(* PLC project LMM.project, Inovance company InoProShop(V1.9.1.6) InoProShop(V1.9.1.6) *)
(* stored: creationDateTime 2026-09-12T22:49:48.5577606, modificationDateTime 2026-09-12T22:49:26.9924488 *)

VAR_GLOBAL  (* GVL *)
  StartBtn AT %IX1.6 : BOOL;  (* 【面板启动】→ HMI_xStart *)
  StopBtn AT %IX1.4 : BOOL;  (* 【面板停止】→ HMI_xStop *)
  ResetBtn : BOOL;  (* 【面板复位】→ HMI_xStopHold3s；地址现场另绑 *)
  EStop AT %IX0.4 : BOOL;  (* 【面板急停】正常=TRUE 按下=FALSE *)
  StopLamp AT %QX0.6 : BOOL;  (* 【停止指示灯】← Dev_xStop *)
  StartLamp AT %QX0.7 : BOOL;  (* 【运行指示灯】← Dev_xRun *)
  JogFwd : BOOL;  (* 【面板前进】手动 X+ *)
  JogBwd : BOOL;  (* 【面板后退】手动 X- *)
  JogRight : BOOL;  (* 【面板右】手动 Y+ *)
  JogLeft : BOOL;  (* 【面板左】手动 Y- *)
  JogUp : BOOL;  (* 【面板上】手动 Z+ *)
  JogDown : BOOL;  (* 【面板下】手动 Z- *)
  JogClockAdd : BOOL;  (* 【面板顺时针】手动 R+ *)
  JogClockMis : BOOL;  (* 【面板逆时针】手动 R- *)
  HMI_xEStop : BOOL;  (* 【急停】TRUE正常 FALSE按下 = 物理 AND 触摸屏Req AND Web *)
  HMI_xStop : BOOL;  (* 【停止】任一源为真即停；长按3s=复位 *)
  HMI_xStopHold3s : BOOL;  (* 【复位】清急停锁存 + 轴故障复位 *)
  HMI_xStart : BOOL;  (* 【启动】上升沿 *)
  HMI_xEnable : BOOL;  (* 【启动别名】与 HMI_xStart 等效 *)
  xEStopLatched : BOOL;  (* 【急停锁存】仅复位可清 *)
  xFaultAggregate : BOOL;  (* 【故障汇总】任轴 ErrorStop *)
  eCtrlSrc : INT;  (* 【控制源】0=面板/触摸屏 1=远程Web；仅 PRG_TcpHmi 写 *)
  eOpMode : INT;  (* 【运行方式】0手动 1自动 *)
  iAlarmID : INT;  (* 【内部报警号】 *)
  HMI_eDevState : INT;  (* 【只读·状态码】0停 1运行 2错误 *)
  HMI_eOpMode : INT;  (* 【只读·方式显示】0手动 1自动 *)
  HMI_iAlarmShow : INT;  (* 【只读·报警号】1001急停 1002轴故障 1005力超时 1006从站失败 1007未就绪；1008已废 *)
  Dev_xStop : BOOL;  (* 【内部·停止派生】 *)
  Dev_xRun : BOOL;  (* 【内部·运行派生】 *)
  Dev_xError : BOOL;  (* 【内部·故障派生】 *)
  HMI_xDevStop : BOOL;  (* 【只读·停止灯】 *)
  HMI_xDevRun : BOOL;  (* 【只读·运行灯】 *)
  HMI_xDevError : BOOL;  (* 【只读·故障灯】 *)
  HMI_xLampEStop : BOOL;  (* 【只读·急停指示】 *)
  HMI_xLampEnableOk : BOOL;  (* 【只读·就绪灯】 *)
  HMI_xLampFault : BOOL;  (* 【只读·故障指示】 *)
  HMI_xAutoMode : BOOL;  (* 【模式】FALSE手动 TRUE自动 *)
  HMI_xJogXPos : BOOL;  (* 【X+】M1=M2 同速同向；与旋转互斥 *)
  HMI_xJogXNeg : BOOL;  (* 【X-】 *)
  HMI_xSpinLeft : BOOL;  (* 【左旋转】差速原地转；与 X± 互斥 *)
  HMI_xSpinRight : BOOL;  (* 【右旋转】 *)
  HMI_xJogYPos : BOOL;  (* 【Y+】受限位 *)
  HMI_xJogYNeg : BOOL;  (* 【Y-】 *)
  HMI_xJogZPos : BOOL;  (* 【Z+】回零后软限位 [-0.7,0] *)
  HMI_xJogZNeg : BOOL;  (* 【Z-】 *)
  HMI_xJogRPos : BOOL;  (* 【R+】需 xM5Ready *)
  HMI_xJogRNeg : BOOL;  (* 【R-】 *)
  HMI_xHomeY : BOOL;  (* 【Y回零】 *)
  HMI_xHomeZ : BOOL;  (* 【Z回零】完成后软限位生效 *)
  HMI_xHomeR : BOOL;  (* 【R回零】编码器回零 *)
  HMI_iHomeAxis : INT := 0;  (* 【回零轴选择】0无 1Y 2Z 3R *)
  HMI_xHomeExec : BOOL;  (* 【回零执行】对选定轴 *)
  HMI_xHomedY : BOOL;  (* 【只读·Y已回零】 *)
  HMI_xHomedZ : BOOL;  (* 【只读·Z已回零】 *)
  HMI_xHomedR : BOOL;  (* 【只读·R已回零】 *)
  HMI_xHomeBusyY : BOOL;  (* 【只读·Y回零中】 *)
  HMI_xHomeBusyZ : BOOL;  (* 【只读·Z回零中】 *)
  HMI_xHomeBusyR : BOOL;  (* 【只读·R回零中】 *)
  HMI_xAutoStart : BOOL;  (* 【自动启动】上升沿 *)
  HMI_xAutoAbort : BOOL;  (* 【自动中止】立即结束 *)
  HMI_rHeadingErr : REAL := 0.0;  (* 【航向误差】视觉/外部纠偏输入（实时量，不保持） *)
  iAutoStep : INT;  (* 【自动步】0Idle..6Done *)
  HMI_iAutoStepShow : INT;  (* 【只读·自动步号】 *)
  HMI_xAutoBusy : BOOL;  (* 【只读·自动忙】 *)
  HMI_xAutoDone : BOOL;  (* 【只读·自动完成】 *)
  Force_xEnable : BOOL := TRUE;  (* 【力通讯总使能】 *)
  Force_wInRaw AT %IW102 : WORD;  (* 组态读通道：0x0000 原始力 *)
  Force_wOutTare AT %QW42 : WORD;  (* 组态写通道：0x0011 去皮 *)
  Force_wOutUnit AT %QW43 : WORD := 5;  (* 组态写通道：0x0002 单位 5=N *)
  Force_rScale : REAL := 0.01;  (* 原始值倍率 *)
  Force_xReadTrig : BOOL;  (* 【内部·力读触发】组态用，勿绑屏 *)
  Force_xCommOk : BOOL;  (* 【只读·力通讯正常】 *)
  Force_xTimeout : BOOL;  (* 【只读·力超时】报警1005 *)
  Force_xSlaveFail : BOOL;  (* 【只读·从站使能失败】报警1006 *)
  Force_xTareBusy : BOOL;  (* 【只读·去皮中】 *)
  Force_xTareDone : BOOL;  (* 【只读·去皮完成】 *)
  Force_iRaw : INT;  (* 【只读·原始计数】 *)
  Force_iState : INT;  (* 【只读·力任务状态】 *)
  rForceAct : REAL;  (* 【实际力】N；Axis 任务写（模拟时 Logic 写） *)
  rForceKp : REAL;  (* 【内部·恒力Kp】 *)
  HMI_rForceSim : REAL;  (* 【力模拟值】N *)
  HMI_xForceSimEnable : BOOL;  (* 【力模拟使能】台架用 *)
  HMI_xForceTare : BOOL;  (* 【去皮】上升沿 *)
  HMI_xForceUntare : BOOL;  (* 【取消去皮】上升沿 *)
  HMI_xForceGuide : BOOL;  (* 【力引导电平】TRUE 持续 Z 恒力跟随 *)
  HMI_rForceShow : REAL;  (* 【只读·显示力】N *)
  Logic_xForceTare : BOOL;  (* 【内部·自动步去皮脉冲】 *)
  I_xLimYPos : BOOL;  (* 【Y正限位开关】 *)
  I_xLimYNeg : BOOL;  (* 【Y负限位开关】 *)
  I_xLimZPos : BOOL;  (* 【Z正限位开关】 *)
  I_xLimZNeg : BOOL;  (* 【Z负限位开关】 *)
  xIlk_BlockYPlus : BOOL;  (* 【联锁禁Y+】开关 ∨ Cfg 限位 *)
  xIlk_BlockYNeg : BOOL;  (* 【联锁禁Y-】 *)
  xIlk_BlockZPlus : BOOL;  (* 【联锁禁Z+】 *)
  xIlk_BlockZNeg : BOOL;  (* 【联锁禁Z-】 *)
  xM5Ready : BOOL := TRUE;  (* 【第5轴就绪】FALSE=忽略 R *)
  AxisCmd_xPower : BOOL;  (* 【轴使能】= 安全条件 *)
  AxisCmd_xStopAll : BOOL;  (* 【全停】急停/停止/故障/中止 *)
  AxisCmd_xResetFault : BOOL;  (* 【故障复位脉冲】 *)
  AxisCmd_xJogXPos : BOOL;  (* 【X+】 *)
  AxisCmd_xJogXNeg : BOOL;  (* 【X-】 *)
  AxisCmd_xSpinLeft : BOOL;  (* 【左旋】 *)
  AxisCmd_xSpinRight : BOOL;  (* 【右旋】 *)
  AxisCmd_xJogYPos : BOOL;  (* 【Y+】 *)
  AxisCmd_xJogYNeg : BOOL;  (* 【Y-】 *)
  AxisCmd_xJogZPos : BOOL;  (* 【Z+】 *)
  AxisCmd_xJogZNeg : BOOL;  (* 【Z-】 *)
  AxisCmd_xJogRPos : BOOL;  (* 【R+】 *)
  AxisCmd_xJogRNeg : BOOL;  (* 【R-】 *)
  AxisCmd_xHomeY : BOOL;  (* 【Y回零】完成/停止清 *)
  AxisCmd_xHomeZ : BOOL;  (* 【Z回零】 *)
  AxisCmd_xHomeR : BOOL;  (* 【R回零】 *)
  AxisCmd_xMoveRelX : BOOL;  (* 【X相对走距】速度模式+里程判完成 *)
  AxisCmd_rMoveDistX : REAL;  (* 【X相对距离】 *)
  AxisCmd_rMoveVelX : REAL;  (* 【X相对速度】 *)
  AxisCmd_xMoveRelY : BOOL;  (* 【Y相对】 *)
  AxisCmd_rMoveDistY : REAL;  (* 【Y相对距离】自动=跨距 *)
  AxisCmd_rMoveVelY : REAL;  (* 【Y速度】 *)
  AxisCmd_xMoveAbsY : BOOL;  (* 【Y绝对】归位用 *)
  AxisCmd_rMoveAbsPosY : REAL;  (* 【Y绝对目标】 *)
  AxisCmd_xForceFollow : BOOL;  (* 【Z力跟随】 *)
  AxisCmd_rForceSet : REAL;  (* 【力目标】 *)
  AxisCmd_rForceKp : REAL;  (* 【力Kp】 *)
  AxisCmd_rForceVelMax : REAL;  (* 【力跟随限速】 *)
  AxisCmd_xHoldR : BOOL;  (* 【R保持角】 *)
  AxisCmd_rRHoldPos : REAL;  (* 【R保持角位置】 *)
  AxisCmd_rHeadingErr : REAL;  (* 【航向误差】 *)
  AxisCmd_rTrackKp : REAL;  (* 【纠偏Kp】 *)
  AxisCmd_rJogVelX : REAL;  (* 【X点动速度】 *)
  AxisCmd_rSpinVel : REAL := 0.0;  (* 【旋转速度】 *)
  AxisCmd_rJogVelY : REAL;  (* 【Y点动速度】 *)
  AxisCmd_rJogVelZ : REAL;  (* 【Z点动速度】 *)
  AxisCmd_rJogVelR : REAL;  (* 【R点动速度】 *)
  AxisCmd_rWheelBase : REAL;  (* 【跨距】限幅 4..6 *)
  AxisCmd_rAccX : REAL;  (* 【X加速度】 *)
  AxisCmd_rDecX : REAL;  (* 【X减速度】 *)
  AxisCmd_rAccY : REAL;  (* 【Y加速度】 *)
  AxisCmd_rDecY : REAL;  (* 【Y减速度】 *)
  AxisCmd_rAccZ : REAL;  (* 【Z加速度】 *)
  AxisCmd_rDecZ : REAL;  (* 【Z减速度】 *)
  AxisCmd_rAccR : REAL;  (* 【R加速度】 *)
  AxisCmd_rDecR : REAL;  (* 【R减速度】 *)
  AxisFb_rVelCmdM1 : REAL;  (* 【只读·M1速度指令】含纠偏/旋转 *)
  AxisFb_rVelCmdM2 : REAL;  (* 【只读·M2速度指令】 *)
  AxisFb_rVelActM1 : REAL;  (* 【只读·M1实际速度】m/s；fbX.rVelActM1Out→状态 word32 *)
  AxisFb_rVelActM2 : REAL;  (* 【只读·M2实际速度】m/s；fbX.rVelActM2Out→状态 word34 *)
  AxisFb_rPosM1 : REAL;  (* 【只读·M1位置】 *)
  AxisFb_rPosM2 : REAL;  (* 【只读·M2位置】 *)
  AxisFb_rPosX : REAL;  (* 【只读·Virtual X 位置】走距判据 *)
  AxisFb_rSyncErr : REAL;  (* 【只读·M1-M2 同步误差】 *)
  AxisFb_rVelFactorX : REAL;  (* 【只读·Virtual Override 倍率】 *)
  AxisFb_xGantryCoupled : BOOL;  (* 【只读·龙门已 GearIn】M1且M2 *)
  AxisFb_xInGearM1 : BOOL;  (* 【只读·M1 电子齿轮 InGear】 *)
  AxisFb_xInGearM2 : BOOL;  (* 【只读·M2 电子齿轮 InGear】 *)
  AxisFb_xPoweredV : BOOL;  (* 【只读·Virtual 已使能】 *)
  AxisFb_xSyncWarn : BOOL;  (* 【只读·同步预警】 *)
  AxisFb_xSyncFault : BOOL;  (* 【只读·同步跳闸】已废，恒 FALSE *)
  AxisFb_iGantryState : INT;  (* 【只读·0Idle 1Coupling 2Coupled 3Decouple 4Diff 5Align】 *)
  AxisFb_rPosY : REAL;  (* 【只读·Y位置】 *)
  AxisFb_rPosZ : REAL;  (* 【只读·Z位置】 *)
  AxisFb_rPosR : REAL;  (* 【只读·R位置/角度】 *)
  AxisFb_xStandstill1 : BOOL;  (* 【只读·M1静止】 *)
  AxisFb_xStandstill2 : BOOL;  (* 【只读·M2静止】 *)
  AxisFb_xStandstillY : BOOL;  (* 【只读·Y静止】 *)
  AxisFb_xStandstillZ : BOOL;  (* 【只读·Z静止】 *)
  AxisFb_xStandstillR : BOOL;  (* 【只读·R静止】 *)
  AxisFb_xMovingM1 : BOOL;  (* 【只读·M1运动中】 *)
  AxisFb_xMovingM2 : BOOL;  (* 【只读·M2运动中】 *)
  AxisFb_xMovingY : BOOL;  (* 【只读·Y运动中】 *)
  AxisFb_xMovingZ : BOOL;  (* 【只读·Z运动中】 *)
  AxisFb_xMovingR : BOOL;  (* 【只读·R运动中】 *)
  AxisFb_xPoweredM1 : BOOL;  (* 【只读·M1已使能】 *)
  AxisFb_xPoweredM2 : BOOL;  (* 【只读·M2已使能】 *)
  AxisFb_xPoweredY : BOOL;  (* 【只读·Y已使能】 *)
  AxisFb_xPoweredZ : BOOL;  (* 【只读·Z已使能】 *)
  AxisFb_xPoweredR : BOOL;  (* 【只读·R已使能】 *)
  AxisFb_xReadyM1 : BOOL;  (* 【只读·M1就绪】 *)
  AxisFb_xReadyM2 : BOOL;  (* 【只读·M2就绪】 *)
  AxisFb_xReadyY : BOOL;  (* 【只读·Y就绪】 *)
  AxisFb_xReadyZ : BOOL;  (* 【只读·Z就绪】 *)
  AxisFb_xReadyR : BOOL;  (* 【只读·R就绪】 *)
  AxisFb_xReady : BOOL;  (* 【只读·全轴就绪】FALSE → 报警1007 *)
  AxisFb_xHomedY : BOOL;  (* 【只读·Y已回零】 *)
  AxisFb_xHomedZ : BOOL;  (* 【只读·Z已回零】 *)
  AxisFb_xHomedR : BOOL;  (* 【只读·R已回零】 *)
  AxisFb_xFaultM1 : BOOL;  (* 【只读·M1故障】 *)
  AxisFb_xFaultM2 : BOOL;  (* 【只读·M2故障】 *)
  AxisFb_xFaultY : BOOL;  (* 【只读·Y故障】 *)
  AxisFb_xFaultZ : BOOL;  (* 【只读·Z故障】 *)
  AxisFb_xFaultR : BOOL;  (* 【只读·R故障】 *)
  AxisFb_xMoveDoneX : BOOL;  (* 【只读·X走距完成】 *)
  AxisFb_xMoveDoneY : BOOL;  (* 【只读·Y完成】 *)
  MB_CmdIn AT %IW103 : ARRAY[0..95] OF WORD;  (* 【命令入】Holding 1000..1095 *)
  MB_StatusOut AT %QW44 : ARRAY[0..95] OF WORD;  (* 【状态出】Holding 1100..1195 *)
  Tcp_iCommStatus : INT;  (* 【只读·通讯诊断】0离线 1在线 2版本错 3序号错 4超时 *)
  Tcp_xConnected : BOOL;  (* 【只读·远程已连接】 *)
  Tcp_xTimeout : BOOL;  (* 【只读·远程超时】 *)
  Tcp_xOnline : BOOL;  (* 【只读·远程在线可用】 *)
  Tcp_wLastHb : WORD;  (* 【内部·上次心跳】 *)
  Tcp_wLastSeq : WORD;  (* 【内部·上次命令序号】 *)
  Tcp_wStatusSeq : WORD;  (* 【内部·状态序号】 *)
  Tcp_xEStop : BOOL := TRUE;  (* 【Web影子·急停】掉线强制 TRUE *)
  Tcp_xStop : BOOL;  (* 【Web影子·停止】 *)
  Tcp_xStopHold3s : BOOL;  (* 【Web影子·复位】 *)
  Tcp_xStart : BOOL;  (* 【Web影子·启动】 *)
  Tcp_xEnable : BOOL;  (* 【Web影子·启动别名】 *)
  Tcp_xAutoMode : BOOL;  (* 【Web影子·模式】 *)
  Tcp_xJogXPos : BOOL;  (* 【Web影子·X+】 *)
  Tcp_xJogXNeg : BOOL;  (* 【Web影子·X-】 *)
  Tcp_xSpinLeft : BOOL;  (* 【Web影子·左旋】 *)
  Tcp_xSpinRight : BOOL;  (* 【Web影子·右旋】 *)
  Tcp_xJogYPos : BOOL;  (* 【Web影子·Y+】 *)
  Tcp_xJogYNeg : BOOL;  (* 【Web影子·Y-】 *)
  Tcp_xJogZPos : BOOL;  (* 【Web影子·Z+】 *)
  Tcp_xJogZNeg : BOOL;  (* 【Web影子·Z-】 *)
  Tcp_xJogRPos : BOOL;  (* 【Web影子·R+】 *)
  Tcp_xJogRNeg : BOOL;  (* 【Web影子·R-】 *)
  Tcp_xHomeY : BOOL;  (* 【Web影子·Y回零】 *)
  Tcp_xHomeZ : BOOL;  (* 【Web影子·Z回零】 *)
  Tcp_xHomeR : BOOL;  (* 【Web影子·R回零】 *)
  Tcp_iHomeAxis : INT := 0;  (* 【Web影子·回零轴选择】 *)
  Tcp_xHomeExec : BOOL;  (* 【Web影子·回零执行】 *)
  Tcp_rJogVelX : REAL := 0.4;  (* 【Web影子·X速度】 *)
  Tcp_rSpinVel : REAL := 0.3;  (* 【Web影子·旋转速度】 *)
  Tcp_rJogVelY : REAL := 0.3;  (* 【Web影子·Y速度】 *)
  Tcp_rJogVelZ : REAL := 0.2;  (* 【Web影子·Z速度】 *)
  Tcp_rJogVelR : REAL := 0.2;  (* 【Web影子·R速度】 *)
  Tcp_xAutoStart : BOOL;  (* 【Web影子·自动启动】 *)
  Tcp_xAutoAbort : BOOL;  (* 【Web影子·自动中止】 *)
  Tcp_rAutoDistX : REAL := 1.0;  (* 【Web影子·自动X距】 *)
  Tcp_rAutoVelX : REAL := 0.4;  (* 【Web影子·自动X速】 *)
  Tcp_rAutoVelY : REAL := 0.3;  (* 【Web影子·自动Y速】 *)
  Tcp_rAutoVelZ : REAL := 0.15;  (* 【Web影子·自动Z速】 *)
  Tcp_rWheelBase : REAL := 5.0;  (* 【Web影子·跨距】 *)
  Tcp_rForceSet : REAL := 100.0;  (* 【Web影子·力设定】 *)
  Tcp_xForceSimEnable : BOOL := FALSE;  (* 【Web影子·力模拟使能】 *)
  Tcp_rForceSim : REAL;  (* 【Web影子·力模拟值】 *)
  Tcp_xForceTare : BOOL;  (* 【Web影子·去皮】 *)
  Tcp_xForceUntare : BOOL;  (* 【Web影子·取消去皮】 *)
  Tcp_xForceGuide : BOOL;  (* 【Web影子·力引导】 *)
  Tcp_iAutoPasses : INT := 1;  (* 【Web影子·自动道数】 *)
  Tcp_rHeadingErr : REAL := 0.0;  (* 【Web影子·航向误差】 *)
  Tcp_rKpTrack : REAL;  (* 【Web影子·纠偏Kp】 *)
  Tcp_rKpForce : REAL;  (* 【Web影子·力Kp】 *)
  Tcp_rAccX : REAL := 100.0;  (* 【Web影子·X加速度】 *)
  Tcp_rDecX : REAL := 100.0;  (* 【Web影子·X减速度】 *)
  Tcp_rAccY : REAL := 100.0;  (* 【Web影子·Y加速度】 *)
  Tcp_rDecY : REAL := 100.0;  (* 【Web影子·Y减速度】 *)
  Tcp_rAccZ : REAL := 100.0;  (* 【Web影子·Z加速度】 *)
  Tcp_rDecZ : REAL := 100.0;  (* 【Web影子·Z减速度】 *)
  Tcp_rAccR : REAL := 100.0;  (* 【Web影子·R加速度】 *)
  Tcp_rDecR : REAL := 100.0;  (* 【Web影子·R减速度】 *)
  HMI_xStartReq : BOOL;  (* 【触摸屏启动】 *)
  HMI_xStopReq : BOOL;  (* 【触摸屏停止】 *)
  HMI_xResetReq : BOOL;  (* 【触摸屏复位】 *)
  HMI_xEStopReq : BOOL := TRUE;  (* 【触摸屏急停】TRUE正常 *)
  HMI_xAutoStartReq : BOOL;  (* 【触摸屏自动启动】 *)
  HMI_xAutoAbortReq : BOOL;  (* 【触摸屏自动中止】 *)
  {attribute 'retain'}
  HMI_rJogVelX : REAL := 0.4;  (* 【X直行速度】与旋转速度分开 *)
  {attribute 'retain'}
  HMI_rSpinVel : REAL := 0.3;  (* 【左右旋速度】 *)
  {attribute 'retain'}
  HMI_rJogVelY : REAL := 0.4;  (* 【Y点动速度】 *)
  {attribute 'retain'}
  HMI_rJogVelZ : REAL := 0.4;  (* 【Z点动速度】力跟随限速后备 *)
  {attribute 'retain'}
  HMI_rJogVelR : REAL := 0.2;  (* 【R点动速度】 *)
  {attribute 'retain'}
  HMI_rAccX : REAL := 25;  (* 【X加速度】 *)
  {attribute 'retain'}
  HMI_rDecX : REAL := 25;  (* 【X减速度】 *)
  {attribute 'retain'}
  HMI_rAccY : REAL := 25;  (* 【Y加速度】 *)
  {attribute 'retain'}
  HMI_rDecY : REAL := 25;  (* 【Y减速度】 *)
  {attribute 'retain'}
  HMI_rAccZ : REAL := 25;  (* 【Z加速度】 *)
  {attribute 'retain'}
  HMI_rDecZ : REAL := 25;  (* 【Z减速度】 *)
  {attribute 'retain'}
  HMI_rAccR : REAL := 25;  (* 【R加速度】 *)
  {attribute 'retain'}
  HMI_rDecR : REAL := 25;  (* 【R减速度】 *)
  {attribute 'retain'}
  HMI_rAutoDistX : REAL := 1.0;  (* 【自动X走距】每道 *)
  {attribute 'retain'}
  HMI_rAutoVelX : REAL := 0.4;  (* 【自动X速度】 *)
  {attribute 'retain'}
  HMI_rAutoVelY : REAL := 0.3;  (* 【自动Y速度】 *)
  {attribute 'retain'}
  HMI_rAutoVelZ : REAL := 0.15;  (* 【自动Z速度】力跟随限速参考 *)
  {attribute 'retain'}
  HMI_rWheelBase : REAL := 5.0;  (* 【龙门跨距=Y行程】4~6 m *)
  {attribute 'retain'}
  HMI_iAutoPasses : INT := 1;  (* 【自动总道数】≥1 *)
  {attribute 'retain'}
  HMI_rForceSet : REAL := 100.0;  (* 【恒力设定】N *)
  {attribute 'retain'}
  HMI_rKpForce : REAL := 1.0;  (* 【力跟随Kp】 *)
  {attribute 'retain'}
  HMI_rKpTrack : REAL := 0.0;  (* 【直线纠偏Kp】 *)
  {attribute 'retain'}
  Cfg_rLimYPos : REAL := 6.0;  (* 【Y正限位】m，默认跨距上限 *)
  {attribute 'retain'}
  Cfg_rLimYNeg : REAL := 0.0;  (* 【Y负限位】m *)
  {attribute 'retain'}
  Cfg_rLimZPos : REAL := 0.0;  (* 【Z正限位】上 *)
  {attribute 'retain'}
  Cfg_rLimZNeg : REAL := -0.7;  (* 【Z负限位】下压行程 *)
  {attribute 'retain'}
  Cfg_rLimRPos : REAL := 180.0;  (* 【R正限位】度 *)
  {attribute 'retain'}
  Cfg_rLimRNeg : REAL := -180.0;  (* 【R负限位】度 *)
  {attribute 'retain'}
  Cfg_rVelBaseMaxX : REAL := 1.0;  (* 【X速度基准】诊断倍率分母；≥最大 Jog/Auto *)
  {attribute 'retain'}
  Cfg_rPhaseMax : REAL := 0.01;  (* 【跟轨相位限幅】u；连续 Phasing *)
  {attribute 'retain'}
  Cfg_rSyncWarn : REAL := 0.02;  (* 【同步预警】|M1-M2|；降速 *)
  {attribute 'retain'}
  Cfg_rSyncFault : REAL := 0.05;  (* 【同步跳闸】已废；保留 RETAIN 布局 *)
  HMI_xDirectEnable : BOOL;  (* 【X直控·Web使能】命令镜像 word5 bit10；与 Vis_xEnable 取或，视觉优先 *)
  HMI_rVelM1Set : REAL;  (* 【X直控·M1设定速度】m/s；命令镜像 word54 (INT×1000) *)
  HMI_rVelM2Set : REAL;  (* 【X直控·M2设定速度】m/s；命令镜像 word55 (INT×1000) *)
  Vis_xEnable : BOOL;  (* 【视觉直控使能】命令镜像 word56 bit0（视觉侧写） *)
  Vis_wSeq : WORD;  (* 【视觉心跳序号】命令镜像 word57；变化即在线，>200ms 不变离线 *)
  Vis_rVelM1Set : REAL;  (* 【视觉直控·M1速度】命令镜像 word58 (INT×1000) *)
  Vis_rVelM2Set : REAL;  (* 【视觉直控·M2速度】命令镜像 word59 (INT×1000) *)
  Direct_xEnable : BOOL;  (* 【X直控·在役】PRG_Logic 仲裁后给 AxisCmd_xDirectVel *)
  Direct_xOnline : BOOL;  (* 【X直控·视觉在线】Vis_wSeq 200ms 内变化 *)
  Direct_wSeqEcho : WORD;  (* 【X直控·视觉序号回显】状态镜像 word31 *)
  Direct_xActive : BOOL;  (* 【X直控·FB在役】状态镜像 word28 bit0 *)
  Direct_rVelM1Act : REAL;  (* 【X直控·M1实际速度】状态镜像 word29 (INT×1000) *)
  Direct_rVelM2Act : REAL;  (* 【X直控·M2实际速度】状态镜像 word30 (INT×1000) *)
  AxisCmd_xDirectVel : BOOL;  (* 【X直控·命令】TRUE=FB_XDual 走 eMode=4 外部直控 *)
  AxisCmd_rVelM1Set : REAL;  (* 【X直控·M1目标速度】m/s *)
  AxisCmd_rVelM2Set : REAL;  (* 【X直控·M2目标速度】m/s *)
  HMI_iDirectModeX : UINT;  (* 【直控·X模式】命令 word60；0idle 1vel（X 仅速度） *)
  HMI_rDirectPosX : REAL;  (* 【直控·X整机目标位置】命令 word61/62 ×1000；整机速度环可选 *)
  HMI_iDirectModeY : UINT;  (* 【直控·Y模式】命令 word63；0idle 1vel 2posAbs 3posRel *)
  HMI_rDirectVelY : REAL;  (* 【直控·Y速度】命令 word64 ×1000；m/s *)
  HMI_rDirectPosY : REAL;  (* 【直控·Y目标位置】命令 word65/66 ×1000；m *)
  HMI_iDirectModeZ : UINT;  (* 【直控·Z模式】命令 word67；0idle 1vel 2posAbs 3posRel *)
  HMI_rDirectVelZ : REAL;  (* 【直控·Z速度】命令 word68 ×1000；m/s *)
  HMI_rDirectPosZ : REAL;  (* 【直控·Z目标位置】命令 word69/70 ×1000；m *)
  HMI_iDirectModeR : UINT;  (* 【直控·R模式】命令 word71；0idle 1vel 2posAbs 3posRel *)
  HMI_rDirectVelR : REAL;  (* 【直控·R速度】命令 word72 ×1000；工程单位/s *)
  HMI_rDirectPosR : REAL;  (* 【直控·R目标位置】命令 word73/74 ×1000；工程单位 *)
  HMI_wDirectSeq : WORD;  (* 【直控·心跳序号】命令 word75；300ms 不变退出直控 *)
  Direct2_xActiveX : BOOL;  (* 【只读·直控·X在役】Logic 写；状态 word42 bit0 *)
  Direct2_xActiveY : BOOL;  (* 【只读·直控·Y在役】Logic 写；状态 word42 bit1 *)
  Direct2_xActiveZ : BOOL;  (* 【只读·直控·Z在役】Logic 写；状态 word42 bit2 *)
  Direct2_xActiveR : BOOL;  (* 【只读·直控·R在役】Logic 写；状态 word42 bit3 *)
  Direct2_xOnline : BOOL;  (* 【只读·直控·心跳在线】Logic 写；状态 word42 bit4 *)
  Direct2_xSafe : BOOL;  (* 【只读·直控·安全允许】Logic 写；状态 word42 bit5 *)
  Direct2_wSeqEcho : WORD;  (* 【只读·直控·心跳回显】Logic 写；状态 word43 *)
  HMI_rForceSetEcho : REAL;  (* 【只读·力设定回显】Logic 写；状态 word44/45 ×100 *)
  AxisFb_rVelActY : REAL;  (* 【只读·Y实际速度】Axis 任务写；状态 word39 ×1000；仅 Axis 任务写 *)
  AxisFb_rVelActZ : REAL;  (* 【只读·Z实际速度】Axis 任务写；状态 word40 ×1000；仅 Axis 任务写 *)
  AxisFb_rVelActR : REAL;  (* 【只读·R实际速度】Axis 任务写；状态 word41 ×1000；仅 Axis 任务写 *)
  AxisCmd_xDirectVelY : BOOL;  (* 【直控·Y速度命令】仅 Logic 写 *)
  AxisCmd_rDirectVelY : REAL;  (* 【直控·Y进给速度】m/s；模式 1 速度，2/3 定位限速 *)
  AxisCmd_xDirectAbsY : BOOL;  (* 【直控·Y绝对命令】仅 Logic 写 *)
  AxisCmd_rDirectAbsY : REAL;  (* 【直控·Y绝对目标】已钳位软限位 *)
  AxisCmd_xDirectRelY : BOOL;  (* 【直控·Y相对命令】仅 Logic 写 *)
  AxisCmd_rDirectRelY : REAL;  (* 【直控·Y相对距离】FB_Servo 内钳位 *)
  AxisCmd_xDirectVelZ : BOOL;  (* 【直控·Z速度命令】仅 Logic 写 *)
  AxisCmd_rDirectVelZ : REAL;  (* 【直控·Z进给速度】m/s *)
  AxisCmd_xDirectAbsZ : BOOL;  (* 【直控·Z绝对命令】仅 Logic 写 *)
  AxisCmd_rDirectAbsZ : REAL;  (* 【直控·Z绝对目标】已钳位软限位 *)
  AxisCmd_xDirectRelZ : BOOL;  (* 【直控·Z相对命令】仅 Logic 写 *)
  AxisCmd_rDirectRelZ : REAL;  (* 【直控·Z相对距离】FB_Servo 内钳位 *)
  AxisCmd_xDirectVelR : BOOL;  (* 【直控·R速度命令】仅 Logic 写 *)
  AxisCmd_rDirectVelR : REAL;  (* 【直控·R进给速度】工程单位/s *)
  AxisCmd_xDirectAbsR : BOOL;  (* 【直控·R绝对命令】仅 Logic 写 *)
  AxisCmd_rDirectAbsR : REAL;  (* 【直控·R绝对目标】已钳位软限位 *)
  AxisCmd_xDirectRelR : BOOL;  (* 【直控·R相对命令】仅 Logic 写 *)
  AxisCmd_rDirectRelR : REAL;  (* 【直控·R相对距离】FB_Servo 内钳位 *)
  Tcp_iDirectModeX : UINT;  (* 【影子·X模式】word60 *)
  Tcp_rDirectPosX : REAL;  (* 【影子·X整机目标】word61/62 ×1000 *)
  Tcp_iDirectModeY : UINT;  (* 【影子·Y模式】word63 *)
  Tcp_rDirectVelY : REAL;  (* 【影子·Y速度】word64 ×1000 *)
  Tcp_rDirectPosY : REAL;  (* 【影子·Y目标】word65/66 ×1000 *)
  Tcp_iDirectModeZ : UINT;  (* 【影子·Z模式】word67 *)
  Tcp_rDirectVelZ : REAL;  (* 【影子·Z速度】word68 ×1000 *)
  Tcp_rDirectPosZ : REAL;  (* 【影子·Z目标】word69/70 ×1000 *)
  Tcp_iDirectModeR : UINT;  (* 【影子·R模式】word71 *)
  Tcp_rDirectVelR : REAL;  (* 【影子·R速度】word72 ×1000 *)
  Tcp_rDirectPosR : REAL;  (* 【影子·R目标】word73/74 ×1000 *)
  Tcp_wDirectSeq : WORD;  (* 【影子·直控心跳】word75 *)
  {attribute 'retain'}
  Cfg_rDirectVelMaxX : REAL := 0.5;  (* 【直控速度上限·X】m/s *)
  {attribute 'retain'}
  Cfg_rDirectVelMaxY : REAL := 0.5;  (* 【直控速度上限·Y】m/s *)
  {attribute 'retain'}
  Cfg_rDirectVelMaxZ : REAL := 0.2;  (* 【直控速度上限·Z】m/s *)
  {attribute 'retain'}
  Cfg_rDirectVelMaxR : REAL := 30.0;  (* 【直控速度上限·R】工程单位/s *)
  {attribute 'retain'}
  Cfg_tDirectTimeout : TIME := TIME#300ms;  (* 【直控看门狗】HMI_wDirectSeq 不变即退出 *)
  HMI_xForcePeakReset : BOOL;  (* 【力峰值复位】TRUE=清零 Force_rPeak（脉冲，命令 word5 bit11） *)
  Force_rPeak : REAL;  (* 【只读·力峰值】N；绝对值峰值，HMI_xForcePeakReset 清零（状态 word46/47 ×100） *)
  Force_wRaw : WORD;  (* 【只读·力原始计数】0..65535，来自 Force_wInRaw（状态 word48） *)
  Tcp_xForcePeakReset : BOOL;  (* 【Web影子·力峰值复位】命令 word5 bit11 *)
  Tcp_rForcePeak : REAL;  (* 【Web影子·力峰值】N；镜像 Force_rPeak *)
  Tcp_wForceRaw : WORD;  (* 【Web影子·力原始计数】镜像 Force_wRaw *)
  AxisFb_rTorqueM1 : REAL;  (* 【只读·M1转矩实际】‰额定转矩（CoE 0x6077 慢速 SDO，1000=100%）；状态 word49 *)
  AxisFb_rTorqueM2 : REAL;  (* 【只读·M2转矩实际】‰额定转矩（CoE 0x6077）；状态 word50 *)
  AxisFb_rCurrentM1 : REAL;  (* 【只读·M1电流实际】‰额定电流（CoE 0x6078）；状态 word51 *)
  AxisFb_rCurrentM2 : REAL;  (* 【只读·M2电流实际】‰额定电流（CoE 0x6078）；状态 word52 *)
  AxisFb_xParamErr : BOOL;  (* 【只读·CoE读取错误】M1/M2 转矩电流 SDO 读失败；状态 word53 bit0 *)
  {attribute 'retain'}
  Cfg_wSdoDevM1 : UINT := 1001;  (* 【CoE SDO 站号·M1】MDX_EC 的 EtherCAT 物理地址（InoProShop 设备树 Address） *)
  {attribute 'retain'}
  Cfg_wSdoDevM2 : UINT := 1002;  (* 【CoE SDO 站号·M2】MDX_EC_1 的 EtherCAT 物理地址 *)
  AxisFb_wSwM1 : WORD;  (* 【只读·M1状态字】CoE 0x6041；状态 word54 *)
  AxisFb_wErrM1 : WORD;  (* 【只读·M1错误码】CoE 0x603F；状态 word55 *)
  AxisFb_wTqMaxM1 : WORD;  (* 【只读·M1最大转矩】CoE 0x6072，0.1%；状态 word56 *)
  AxisFb_wLimPM1 : WORD;  (* 【只读·M1正向转矩限】CoE 0x60E0；状态 word57 *)
  AxisFb_wLimNM1 : WORD;  (* 【只读·M1反向转矩限】CoE 0x60E1；状态 word58 *)
  AxisFb_wSwM2 : WORD;  (* 【只读·M2状态字】CoE 0x6041；状态 word59 *)
  AxisFb_wErrM2 : WORD;  (* 【只读·M2错误码】CoE 0x603F；状态 word60 *)
  AxisFb_wTqMaxM2 : WORD;  (* 【只读·M2最大转矩】CoE 0x6072；状态 word61 *)
  AxisFb_wLimPM2 : WORD;  (* 【只读·M2正向转矩限】CoE 0x60E0；状态 word62 *)
  AxisFb_wLimNM2 : WORD;  (* 【只读·M2反向转矩限】CoE 0x60E1；状态 word63 *)
  AxisFb_wModeM1 : WORD;  (* 【只读·M1运行模式】CoE 0x6060（9=CSV/8=CSP）；状态 word64 *)
  AxisFb_wTq03M1 : WORD;  (* 【只读·M1转矩限值】CoE 0x2403；状态 word65 *)
  AxisFb_wTq04M1 : WORD;  (* 【只读·M1转矩限值】CoE 0x2404；状态 word66 *)
  AxisFb_wTq05M1 : WORD;  (* 【只读·M1转矩限值】CoE 0x2405；状态 word67 *)
  AxisFb_wTq06M1 : WORD;  (* 【只读·M1转矩限值】CoE 0x2406；状态 word68 *)
  AxisFb_wModeM2 : WORD;  (* 【只读·M2运行模式】CoE 0x6060；状态 word69 *)
  AxisFb_wTq03M2 : WORD;  (* 【只读·M2转矩限值】CoE 0x2403；状态 word70 *)
  AxisFb_wTq04M2 : WORD;  (* 【只读·M2转矩限值】CoE 0x2404；状态 word71 *)
  AxisFb_wTq05M2 : WORD;  (* 【只读·M2转矩限值】CoE 0x2405；状态 word72 *)
  AxisFb_wTq06M2 : WORD;  (* 【只读·M2转矩限值】CoE 0x2406；状态 word73 *)
  {attribute 'retain'}
  Cfg_xForceCsvX : BOOL := TRUE;  (* 【0.74 强制 X 双驱 CSV 速度模式】空闲时切 SMC_velocity(0x6060=9) *)
  AxisFb_xModeCsvM1 : BOOL;  (* 【只读·M1 已切 CSV】状态 word74 bit0 *)
  AxisFb_xModeCsvErrM1 : BOOL;  (* 【只读·M1 切 CSV 失败】状态 word74 bit1 *)
  AxisFb_xModeCsvM2 : BOOL;  (* 【只读·M2 已切 CSV】状态 word74 bit2 *)
  AxisFb_xModeCsvErrM2 : BOOL;  (* 【只读·M2 切 CSV 失败】状态 word74 bit3 *)
END_VAR

FUNCTION_BLOCK FB_XDual
  VAR_INPUT
    xEnable : BOOL;
    xStop : BOOL;
    xResetFault : BOOL;
    xJogPos : BOOL;
    xJogNeg : BOOL;
    xSpinLeft : BOOL;
    xSpinRight : BOOL;
    xMoveRel : BOOL;
    rMoveDist : REAL;
    rMoveVel : REAL;
    rJogVel : REAL;
    rSpinVel : REAL;
    rHeadingErr : REAL;
    rKpTrack : REAL;
    rAcc : REAL;
    rDec : REAL;
    rTrimMax : REAL;
    xSyncEnable : BOOL := TRUE;
    rRatioM1 : REAL := 1.0;
    rRatioM2 : REAL := 1.0;
    rHeadingDeadband : REAL := 0.003;
    rTrimFilterTc : REAL := 0.05;
    rCycleSec : REAL := 0.004;
    xDirectMode : BOOL;
    rVelM1Direct : REAL;
    rVelM2Direct : REAL;
    tDirectRetrig : TIME := TIME#40ms;
    wSdoDevM1 : UINT;
    wSdoDevM2 : UINT;
    xForceCsv : BOOL;
  END_VAR
  VAR_OUTPUT
    xMoveDone : BOOL;
    rPosV : REAL;
    rSyncErr : REAL;
    rVelFactor : REAL;
    xCoupled : BOOL;
    xInGearM1 : BOOL;
    xInGearM2 : BOOL;
    xPoweredV : BOOL;
    xSyncWarn : BOOL;
    xSyncFault : BOOL;
    iState : INT;
    iHoldState : INT;
    eSlaveMode : INT;
    rVelCmdM1 : REAL;
    rVelCmdM2 : REAL;
    rPosM1 : REAL;
    rPosM2 : REAL;
    xMovingM1 : BOOL;
    xMovingM2 : BOOL;
    xStandstillM1 : BOOL;
    xStandstillM2 : BOOL;
    xPoweredM1 : BOOL;
    xPoweredM2 : BOOL;
    xReadyM1 : BOOL;
    xReadyM2 : BOOL;
    xFaultM1 : BOOL;
    xFaultM2 : BOOL;
    xVelReqM1 : BOOL;
    xVelReqM2 : BOOL;
    xVelBusyM1 : BOOL;
    xVelBusyM2 : BOOL;
    xErrPowerM1 : BOOL;
    xErrPowerM2 : BOOL;
    xErrVelM1 : BOOL;
    xErrVelM2 : BOOL;
    xVelExecM1 : BOOL;
    xVelExecM2 : BOOL;
    xVelInVelM1 : BOOL;
    xVelInVelM2 : BOOL;
    iVelExecRise : INT;
    rVelActM1Out : REAL;
    rVelActM2Out : REAL;
    xDirectActive : BOOL;
    rTorqueActM1 : REAL;
    rTorqueActM2 : REAL;
    rCurrentActM1 : REAL;
    rCurrentActM2 : REAL;
    xParamErr : BOOL;
    wSwM1 : WORD;
    wErrM1 : WORD;
    wTqMaxM1 : WORD;
    wLimPM1 : WORD;
    wLimNM1 : WORD;
    wSwM2 : WORD;
    wErrM2 : WORD;
    wTqMaxM2 : WORD;
    wLimPM2 : WORD;
    wLimNM2 : WORD;
    wModeM1 : WORD;
    wTq03M1 : WORD;
    wTq04M1 : WORD;
    wTq05M1 : WORD;
    wTq06M1 : WORD;
    wModeM2 : WORD;
    wTq03M2 : WORD;
    wTq04M2 : WORD;
    wTq05M2 : WORD;
    wTq06M2 : WORD;
    xModeCsvM1 : BOOL;
    xModeCsvErrM1 : BOOL;
    xModeCsvM2 : BOOL;
    xModeCsvErrM2 : BOOL;
  END_VAR
  VAR
    fbPowerM1 : MC_Power;
    fbPowerM2 : MC_Power;
    fbResetM1 : MC_Reset;
    fbResetM2 : MC_Reset;
    fbVelM1 : MC_MoveVelocity;
    fbVelM2 : MC_MoveVelocity;
    fbHaltM1 : MC_Halt;
    fbHaltM2 : MC_Halt;
    fbStopM1 : MC_Stop;
    fbStopM2 : MC_Stop;
    fbSdoTqM1 : ETC_CO_SdoRead;
    fbSdoCurM1 : ETC_CO_SdoRead;
    fbSdoSwM1 : ETC_CO_SdoRead;
    fbSdoErrM1 : ETC_CO_SdoRead;
    fbSdoTqMaxM1 : ETC_CO_SdoRead;
    fbSdoLimPM1 : ETC_CO_SdoRead;
    fbSdoLimNM1 : ETC_CO_SdoRead;
    fbSdoModeM1 : ETC_CO_SdoRead;
    fbSdoTq03M1 : ETC_CO_SdoRead;
    fbSdoTq04M1 : ETC_CO_SdoRead;
    fbSdoTq05M1 : ETC_CO_SdoRead;
    fbSdoTq06M1 : ETC_CO_SdoRead;
    fbSdoTqM2 : ETC_CO_SdoRead;
    fbSdoCurM2 : ETC_CO_SdoRead;
    fbSdoSwM2 : ETC_CO_SdoRead;
    fbSdoErrM2 : ETC_CO_SdoRead;
    fbSdoTqMaxM2 : ETC_CO_SdoRead;
    fbSdoLimPM2 : ETC_CO_SdoRead;
    fbSdoLimNM2 : ETC_CO_SdoRead;
    fbSdoModeM2 : ETC_CO_SdoRead;
    fbSdoTq03M2 : ETC_CO_SdoRead;
    fbSdoTq04M2 : ETC_CO_SdoRead;
    fbSdoTq05M2 : ETC_CO_SdoRead;
    fbSdoTq06M2 : ETC_CO_SdoRead;
    abyTqM1 : ARRAY[0..1] OF BYTE;
    abyCurM1 : ARRAY[0..1] OF BYTE;
    abySwM1 : ARRAY[0..1] OF BYTE;
    abyErrM1 : ARRAY[0..1] OF BYTE;
    abyTqMaxM1 : ARRAY[0..1] OF BYTE;
    abyLimPM1 : ARRAY[0..1] OF BYTE;
    abyLimNM1 : ARRAY[0..1] OF BYTE;
    abyModeM1 : ARRAY[0..1] OF BYTE;
    abyTq03M1 : ARRAY[0..1] OF BYTE;
    abyTq04M1 : ARRAY[0..1] OF BYTE;
    abyTq05M1 : ARRAY[0..1] OF BYTE;
    abyTq06M1 : ARRAY[0..1] OF BYTE;
    abyTqM2 : ARRAY[0..1] OF BYTE;
    abyCurM2 : ARRAY[0..1] OF BYTE;
    abySwM2 : ARRAY[0..1] OF BYTE;
    abyErrM2 : ARRAY[0..1] OF BYTE;
    abyTqMaxM2 : ARRAY[0..1] OF BYTE;
    abyLimPM2 : ARRAY[0..1] OF BYTE;
    abyLimNM2 : ARRAY[0..1] OF BYTE;
    abyModeM2 : ARRAY[0..1] OF BYTE;
    abyTq03M2 : ARRAY[0..1] OF BYTE;
    abyTq04M2 : ARRAY[0..1] OF BYTE;
    abyTq05M2 : ARRAY[0..1] OF BYTE;
    abyTq06M2 : ARRAY[0..1] OF BYTE;
    fbSetModeM1 : SMC_SetControllerMode;
    fbSetModeM2 : SMC_SetControllerMode;
    xModeVelDoneM1 : BOOL;
    xModeVelDoneM2 : BOOL;
    fbWrModeM1 : ETC_CO_SdoWrite4;
    fbWrModeM2 : ETC_CO_SdoWrite4;
    xModeReqM1 : BOOL;
    xModeReqM2 : BOOL;
    abyModeWr : ARRAY[1..4] OF BYTE;
    xModeWrDoneM1 : BOOL;
    xModeWrDoneM2 : BOOL;
    xModeWrErrM1 : BOOL;
    xModeWrErrM2 : BOOL;
    wSdoRaw : WORD;
    tonSdoSlot : TON;
    iSdoSlot : INT;
    eDirM1 : MC_DIRECTION;
    eDirM2 : MC_DIRECTION;
    eMode : INT;
    eModePrev : INT;
    rBase : REAL;
    rVelActM1 : REAL;
    rVelActM2 : REAL;
    rTrim : REAL;
    rTrimRaw : REAL;
    rTrimFiltered : REAL;
    rAlphaFilter : REAL;
    rUseRatioM1 : REAL;
    rUseRatioM2 : REAL;
    rSyncExpect : REAL;
    rSyncResid : REAL;
    rCorrPos : REAL;
    rCorrV1 : REAL;
    rCorrV2 : REAL;
    rVelFF1 : REAL;
    rVelFF2 : REAL;
    rKpSync : REAL := 0.05;
    rKvSync : REAL := 0.0;
    rSyncDeadband : REAL := 0.02;
    rCorrPosMax : REAL := 0.08;
    rCorrVelMax : REAL := 0.06;
    xStraightEdge : BOOL;
    xJogRaw : BOOL;
    xJogHeld : BOOL;
    tonJogOff : TON;
    tonStillM1 : TON;
    tonStillM2 : TON;
    tonHoldFallback : TON;
    tonJogGrace : TON;
    rHoldVelMax : REAL := 0.5;
    xSoftHold : BOOL;
    xSoftHoldPrev : BOOL;
    xSoftHoldLatched : BOOL;
    fbSetPosM1 : MC_SetPosition;
    fbSetPosM2 : MC_SetPosition;
    xZeroGate : BOOL;
    tonZeroDelay : TON;
    xZeroReady : BOOL;
    xZeroPulsePrev : BOOL;
    xSetPosReq : BOOL;
    xPosZeroed : BOOL;
    xErrSetPosM1 : BOOL;
    xErrSetPosM2 : BOOL;
    xResetEdge : BOOL;
    xResetPrev : BOOL;
    xDirFlipM1 : BOOL;
    xDirFlipM2 : BOOL;
    xVelRunPrevM1 : BOOL;
    xVelRunPrevM2 : BOOL;
    rVelInPrevM1 : REAL;
    rVelInPrevM2 : REAL;
    rVelAppl : REAL;
    rAccUse : REAL;
    rDecUse : REAL;
    rAccLatch : REAL;
    rDecLatch : REAL;
    rVelLatchM1 : REAL;
    rVelLatchM2 : REAL;
    xExecPrev : BOOL;
    rAccSoftMin : REAL := 0.05;
    rAccSoft : REAL;
    rDecSoft : REAL;
    rRampAccMax : REAL := 1.0;
    xDecelActive : BOOL;
    xDecelDone : BOOL;
    rDecelDist : REAL;
    xM1Decel : BOOL;
    xM2Decel : BOOL;
    xBothPowered : BOOL;
    xPowerGate : BOOL;
    xReqVelM1 : BOOL;
    xReqVelM2 : BOOL;
    xNeedHaltM1 : BOOL;
    xNeedHaltM2 : BOOL;
    xRegOn : BOOL;
    xRegOnPrev : BOOL;
    xStopping : BOOL;
    xWasStopping : BOOL;
    xHaltTrig : BOOL;
    xHaltPrev : BOOL;
    xPowerSettled : BOOL;
    xStartReady : BOOL;
    xStopFallback : BOOL;
    tonHaltWin : TON;
    tonPowerOk : TON;
    tonVelHold : TON;
    tonRampLock : TON;
    tonTrimRetrig : TON;
    xTrimWant : BOOL;
    xTrimPulse : BOOL;
    xTrimPulsePrev : BOOL;
    xMoveRelDecelTrig : BOOL;
    xExecM1 : BOOL;
    xExecHold : BOOL;
    xHaltBusy : BOOL;
    xExecBoth : BOOL;
    xDirFlipAny : BOOL;
    xVelHoldOff : BOOL;
    xErrVelPrev : BOOL;
    xRampLock : BOOL;
    rVelFbM1 : REAL;
    rVelFbM2 : REAL;
    rVelFbHoldM1 : REAL;
    rVelFbHoldM2 : REAL;
    rCorrLim : REAL;
    xMovePrev : BOOL;
    xArmed : BOOL;
    rStart : REAL;
    rAvg : REAL;
    rSyncWarnLevel : REAL := 0.05;
    rSyncFaultLevel : REAL := 0.15;
    tonSyncFault : TON;
    tonDirectRetrig : TON;
    xDirectWant : BOOL;
    xDirectPulse : BOOL;
    xDirectPulsePrev : BOOL;
    xHaltDemand : BOOL;
  END_VAR
  VAR_IN_OUT
    AxisM1 : AXIS_REF_SM3;
    AxisM2 : AXIS_REF_SM3;
  END_VAR

            (* ==============================================================================
 * FB_XDual — X 轴双驱（g 线 0.59）：单沿起步 + SM3 斜坡 + Halt 对称减速
 * 铁律：X 轴只经本 FB；FB_Servo 不得持有 X 轴实例。
 *
 *   0.44 根因：Enable 和调节器一起关 → Power FB 停转，驱动收不到卸使能；
 *   运动中切使能 + 刚上使能就 Execute → 连冲、Error 锁死第二次点动。
 *   对齐 FB_Servo：Enable 保持，bRegulatorOn/bDriveStart 跟 xRegOn；
 *   松手 Halt 脉冲刹停，双轴 standstill 后才卸调节器；2s 未静止改发 Stop。
 *   冷启动等 Status 约 80ms 且双轴 standstill 再出速度；短窗内再按不再等。
 *   0.47：禁止 300ms 超时在减速中卸使能（运动中送掉使能报错）。
 *   0.50：幅值差速不撤 Execute。必须重触发的只有换向。
 *   0.51：0.50 仍三次过冲——使能后 20ms 就 Execute（失败连打）+ 爬坡每拍改 Velocity。
 *         上使能后等 Status 80ms；Error 锁 150ms；爬坡只吃基速，到速后再跟 trim。
 *   0.52：xErrVel 不跳仍冲三次+忽快忽慢。根因是 0.51 把 xPowerSettled 绑在 standstill：
 *         轴一动就掉 Execute，松手前 Acc/Dec 反复爬。闭锁一次后保持；残差 P 降增益。
 *   0.53：xVelReq 一直 TRUE 仍冲三次。请求≠Execute；Acc=Jog 时 SM3 梯形拐点 + 使能冲击叠成三次。
 *         PLC 按用户 Acc 爬 FB 速度，SM3 Acc 抬到 ≥10 只负责跟上；松手仍 Halt。
 *   0.54：0.53 不过冲也不走。本机 Execute 保持时 Velocity 不刷新，第一拍 ~0 被锁死。
 *         上升沿一次写入目标速度 + 用户 Acc；爬坡中不改输入；到速后再跟 trim。
 *   0.55：三次过冲=Execute 被拉了三次。PRG_Logic 先清 AxisCmd 再置位，ETHERCAT(prio0)
 *         在 FALSE 空窗采到松手→Halt→再加速。第一次点动 Logic 超时约 3 拍。去抖+一次写入。
 *   0.56：偶发三次过冲。0.55 去抖保了 eMode，但 Power.Status 闪一下仍清 xStartReady，
 *         Execute 掉、锁存清 0，再启动就是又一次过冲。点动中 Execute 闭锁到松开。
 *   0.57：现场仍每次起步沿 X 往复冲 3 次（约 3s）。根因：起步=速度阶跃（Acc=25）
 *         打进 CSV 速度环，激起双驱耦合龙门 ~1Hz 纵向共振。0.53 阶梯爬速本可消过冲，
 *         但本机 Execute 保持时 Velocity 不刷新，首拍 ~0 锁死（"不过冲也不走"）。
 *   0.58：恢复 rVelSlew 阶梯爬速；爬坡期 Execute 每步重触发（OFF/ON 交替一拍，
 *         上升沿重采样）；斜率取用户 Acc/Dec 钳 [0.05, rRampAccMax]，SM3 Acc 只跟梯；
 *         松手/到位先阶梯降到 ~0 再 Halt；MoveRel 剩余≤slew²/2Dec 提前减速；
 *         到位锁 xDecelDone 禁停稳后重爬目标。
 *   0.59：0.58 每步重触发 = 250Hz 沿风暴，现场 acc=0.8 起步仍快速冲 2 次（~1s）、
 *         第三次慢、停死；M2 明显慢于 M1（两侧接受沿时刻不一致，M2 漏沿爬速落后）。
 *         改单沿起步：一个上升沿写最终目标 + 钳制用户 Acc/Dec（0.05~1.0），
 *         SM3 自带斜坡 0→目标（0.8 → 0.5s）；稳态 trim/sync 更新走限频重触发
 *         （≥200ms 一次、差值≥0.004）；减速统一 Halt（用户 Dec 对称）。
 * ============================================================================== *)

rVelFactor := 0.0;
xCoupled := FALSE;
xInGearM1 := FALSE;
xInGearM2 := FALSE;
xPoweredV := FALSE;
eSlaveMode := 0;

(* ------------------- 1. 模式 ------------------- *)
(* 点动 FALSE 短于 40ms 视为空窗，不 Halt、不撤 Execute *)
xJogRaw := (xJogPos XOR xJogNeg) OR xMoveRel;
tonJogOff(IN := xJogHeld AND NOT xJogRaw AND xEnable AND NOT xStop
           AND NOT (xSpinLeft XOR xSpinRight), PT := T#40MS);
IF xStop OR NOT xEnable THEN
    eMode := 0;
    rBase := 0.0;
    xJogHeld := FALSE;
ELSIF xSpinLeft XOR xSpinRight THEN
    IF xSpinLeft THEN
        eMode := 2;
    ELSE
        eMode := 3;
    END_IF;
    rBase := 0.0;
    xJogHeld := FALSE;
ELSIF xDirectMode THEN
    (* 0.60 外部直控优先于点动：视觉接管期间忽略点动/走距输入 *)
    eMode := 4;
    rBase := 0.0;
    xJogHeld := FALSE;
ELSIF xJogRaw THEN
    eMode := 1;
    xJogHeld := TRUE;
    IF xMoveRel THEN
        IF rMoveDist >= 0.0 THEN
            rBase := ABS(rMoveVel);
        ELSE
            rBase := -ABS(rMoveVel);
        END_IF;
    ELSIF xJogPos THEN
        rBase := ABS(rJogVel);
    ELSE
        rBase := -ABS(rJogVel);
    END_IF;
ELSIF xJogHeld AND NOT tonJogOff.Q THEN
    eMode := 1;
ELSE
    eMode := 0;
    rBase := 0.0;
    xJogHeld := FALSE;
END_IF;
iState := eMode;
xStraightEdge := (eMode = 1) AND (eModePrev <> 1);

(* ------------------- 2. 回读 + SoftHold ------------------- *)
rPosM1 := LREAL_TO_REAL(AxisM1.fActPosition);
rPosM2 := LREAL_TO_REAL(AxisM2.fActPosition);
rVelActM1 := LREAL_TO_REAL(AxisM1.fActVelocity);
rVelActM2 := LREAL_TO_REAL(AxisM2.fActVelocity);
rAvg := (rPosM1 + rPosM2) * 0.5;
rPosV := rAvg;
rSyncErr := rPosM1 - rPosM2;

xStandstillM1 := AxisM1.nAxisState = SMC_AXIS_STATE.standstill;
xStandstillM2 := AxisM2.nAxisState = SMC_AXIS_STATE.standstill;
xMovingM1 := (NOT xStandstillM1) OR (ABS(rVelActM1) > 0.01);
xMovingM2 := (NOT xStandstillM2) OR (ABS(rVelActM2) > 0.01);

tonStillM1(IN := NOT xMovingM1, PT := T#200MS);
tonStillM2(IN := NOT xMovingM2, PT := T#200MS);
tonHoldFallback(IN := (eMode = 0) AND NOT xStop AND xEnable
                    AND (ABS(rVelActM1) < rHoldVelMax) AND (ABS(rVelActM2) < rHoldVelMax),
                PT := T#2S);
IF xStop OR NOT xEnable OR (eMode <> 0) THEN
    iHoldState := 0;
    xSoftHoldLatched := FALSE;
ELSIF xSoftHoldLatched THEN
    iHoldState := 2;
ELSIF (tonStillM1.Q AND tonStillM2.Q) OR tonHoldFallback.Q THEN
    iHoldState := 2;
    xSoftHoldLatched := TRUE;
ELSE
    iHoldState := 1;
END_IF;
xSoftHold := iHoldState = 2;
xSoftHoldPrev := xSoftHold;
(* 再按起步 300ms 内隐藏 SoftHold/Halt 残留 bError，避免 Fault→StopAll 发肉 *)
tonJogGrace(IN := (eMode <> 0), PT := T#300MS);

xSyncWarn := ABS(rSyncErr) > rSyncWarnLevel;
tonSyncFault(IN := ABS(rSyncErr) > rSyncFaultLevel, PT := T#500MS);
IF tonSyncFault.Q THEN
    xSyncFault := TRUE;
END_IF;

(* ------------------- 3. 复位仅手动 ------------------- *)
fbResetM1(Axis := AxisM1, Execute := xResetFault);
fbResetM2(Axis := AxisM2, Execute := xResetFault);
IF xResetFault THEN
    xSyncFault := FALSE;
END_IF;

(* ------------------- 4. 使能：Power.Enable 常开，只切调节器 ------------------- *)
(* 松手保持调节器直到双轴 standstill。300ms 超时会在减速未完时卸使能（0.46 报错）。 *)
xWasStopping := xStopping;
IF xStop OR NOT xEnable THEN
    xStopping := FALSE;
ELSIF eMode <> 0 THEN
    xStopping := FALSE;
ELSIF xRegOnPrev THEN
    xStopping := TRUE;
END_IF;
tonHaltWin(IN := xStopping AND (eMode = 0) AND xEnable AND NOT xStop, PT := T#2S);
IF xStopping AND (eMode = 0) AND xStandstillM1 AND xStandstillM2 THEN
    xStopping := FALSE;
END_IF;
xRegOn := xEnable AND NOT xStop AND ((eMode <> 0) OR xStopping);
xStopFallback := xStopping AND tonHaltWin.Q AND NOT (xStandstillM1 AND xStandstillM2) AND NOT xDecelActive;
(* Enable 恒 TRUE，卸使能只走调节器（对齐 FB_Servo；0.44 关 Enable 导致驱动收不到） *)
fbPowerM1(Axis := AxisM1, Enable := TRUE,
          bRegulatorOn := xRegOn, bDriveStart := xRegOn);
fbPowerM2(Axis := AxisM2, Enable := TRUE,
          bRegulatorOn := xRegOn, bDriveStart := xRegOn);

xPoweredM1 := fbPowerM1.Status;
xPoweredM2 := fbPowerM2.Status;
xFaultM1 := AxisM1.bError AND xRegOn AND NOT (xSoftHold OR (iHoldState = 1) OR xStopping OR ((eMode <> 0) AND NOT tonJogGrace.Q));
xFaultM2 := AxisM2.bError AND xRegOn AND NOT (xSoftHold OR (iHoldState = 1) OR xStopping OR ((eMode <> 0) AND NOT tonJogGrace.Q));
(* 就绪 = 使能已给且无故障；不含 xStop / xPowered：
   停止、或按需关调节器(xRegOn=FALSE, 静态)时仍报就绪，避免 Logic 1007 误报。 *)
xReadyM1 := xEnable AND NOT xFaultM1;
xReadyM2 := xEnable AND NOT xFaultM2;
xBothPowered := xPoweredM1 AND xPoweredM2;
xPowerGate := xEnable AND NOT xStop AND NOT xFaultM1 AND NOT xFaultM2;
tonPowerOk(IN := xRegOn AND xBothPowered AND (eMode <> 0), PT := T#80MS);
(* 冷启动闭锁一次。Status 闪烁不得清 xStartReady，否则 Execute 掉了再爬。 *)
IF (eMode = 0) OR NOT xRegOn OR xStop THEN
    xStartReady := FALSE;
ELSIF xWasStopping OR xExecHold THEN
    xStartReady := TRUE;
ELSIF tonPowerOk.Q AND xStandstillM1 AND xStandstillM2 THEN
    xStartReady := TRUE;
END_IF;
xPowerSettled := xRegOn AND (eMode <> 0) AND xStartReady
                 AND (xBothPowered OR xExecHold);

(* 置零：点动/短窗禁止；空闲自动置零会和 Halt 抢轴，只保留手动 Reset *)
IF (eMode <> 0) OR xStopping OR xStop OR NOT xEnable THEN
    xSetPosReq := FALSE;
END_IF;
xZeroGate := FALSE;
tonZeroDelay(IN := FALSE, PT := T#300MS);
xZeroReady := FALSE;
xZeroPulsePrev := FALSE;
xResetEdge := xResetFault AND NOT xResetPrev;
xResetPrev := xResetFault;
IF xResetEdge AND (eMode = 0) AND NOT xStopping THEN
    xSetPosReq := TRUE;
END_IF;
fbSetPosM1(Axis := AxisM1, Execute := xSetPosReq AND (eMode = 0) AND NOT xStopping, Position := 0.0);
fbSetPosM2(Axis := AxisM2, Execute := xSetPosReq AND (eMode = 0) AND NOT xStopping, Position := 0.0);
xErrSetPosM1 := fbSetPosM1.Error;
xErrSetPosM2 := fbSetPosM2.Error;
IF xSetPosReq THEN
    IF (fbSetPosM1.Done AND fbSetPosM2.Done) OR fbSetPosM1.Error OR fbSetPosM2.Error THEN
        xSetPosReq := FALSE;
        xPosZeroed := TRUE;
    END_IF;
END_IF;

(* ------------------- 6. 基速跟手 + 视觉差速 ------------------- *)
rAccUse := ABS(rAcc);
IF rAccUse < rAccSoftMin THEN
    rAccUse := rAccSoftMin;
END_IF;
rDecUse := ABS(rDec);
IF rDecUse < rAccSoftMin THEN
    rDecUse := rAccSoftMin;
END_IF;

(* 0.59：SM3 斜坡用钳制 Acc/Dec（0.05~rRampAccMax）。HMI 25/100 兜底不再变阶跃；
   rDecUse 保留软下限继续供 Stop 急停。 *)
rAccSoft := ABS(rAcc);
IF rAccSoft < rAccSoftMin THEN
    rAccSoft := rAccSoftMin;
END_IF;
IF rAccSoft > rRampAccMax THEN
    rAccSoft := rRampAccMax;
END_IF;
rDecSoft := ABS(rDec);
IF rDecSoft < rAccSoftMin THEN
    rDecSoft := rAccSoftMin;
END_IF;
IF rDecSoft > rRampAccMax THEN
    rDecSoft := rRampAccMax;
END_IF;

(* 0.36：禁止 PLC 再爬 rVelAppl。按下即目标速度，松开即 0，停靠 Halt。 *)
(* 0.59 注：rVelAppl 是最终目标；起步斜坡由 SM3 按 rAccSoft 生成（单沿锁存）。 *)
IF (eMode = 0) OR xStop OR NOT xEnable THEN
    rVelAppl := 0.0;
ELSIF eMode = 1 THEN
    rVelAppl := rBase;
ELSE
    rVelAppl := 0.0;
END_IF;

(* 视觉：同一条基速上 ±trim，不是第二次运动，不撤 Execute *)
rTrimRaw := 0.0;
rCorrPos := 0.0;
rCorrV1 := 0.0;
rCorrV2 := 0.0;
rUseRatioM1 := rRatioM1;
IF rUseRatioM1 < 0.1 THEN
    rUseRatioM1 := 0.1;
END_IF;
rUseRatioM2 := rRatioM2;
IF rUseRatioM2 < 0.1 THEN
    rUseRatioM2 := 0.1;
END_IF;
IF eMode = 1 THEN
    IF ABS(rHeadingErr) > ABS(rHeadingDeadband) THEN
        IF rHeadingErr > 0.0 THEN
            rTrimRaw := (rHeadingErr - ABS(rHeadingDeadband)) * rKpTrack;
        ELSE
            rTrimRaw := (rHeadingErr + ABS(rHeadingDeadband)) * rKpTrack;
        END_IF;
        rTrimRaw := LIMIT(-ABS(rTrimMax), rTrimRaw, ABS(rTrimMax));
    END_IF;
    IF rTrimFilterTc > 0.001 THEN
        rAlphaFilter := rCycleSec / (rTrimFilterTc + rCycleSec);
        rTrimFiltered := rTrimFiltered + rAlphaFilter * (rTrimRaw - rTrimFiltered);
    ELSE
        rTrimFiltered := rTrimRaw;
    END_IF;
    rTrim := rTrimFiltered;
    IF xStraightEdge THEN
        rSyncExpect := rPosM1 - rPosM2;
        rTrimFiltered := 0.0;
        rTrim := 0.0;
        xRampLock := TRUE;
    END_IF;
    rSyncExpect := rSyncExpect + (2.0 * rTrim * rCycleSec);
    rSyncResid := (rPosM1 - rPosM2) - rSyncExpect;
    rCorrLim := ABS(rCorrPosMax);
    IF ABS(rVelAppl) > 0.001 THEN
        IF (0.25 * ABS(rVelAppl)) < rCorrLim THEN
            rCorrLim := 0.25 * ABS(rVelAppl);
        END_IF;
    END_IF;
    IF xSyncEnable AND (ABS(rVelAppl) > 0.001) THEN
        IF ABS(rSyncResid) > rSyncDeadband THEN
            rCorrPos := LIMIT(-rCorrLim, rKpSync * rSyncResid, rCorrLim);
        END_IF;
        rCorrV1 := LIMIT(-ABS(rCorrVelMax), rKvSync * ((rVelAppl + rTrim) - rVelActM1), ABS(rCorrVelMax));
        rCorrV2 := LIMIT(-ABS(rCorrVelMax), rKvSync * ((rVelAppl - rTrim) - rVelActM2), ABS(rCorrVelMax));
    END_IF;
    rVelFF1 := rVelAppl + rTrim;
    rVelFF2 := rVelAppl - rTrim;
    rVelCmdM1 := (rVelFF1 - 0.5 * rCorrPos + rCorrV1) * rUseRatioM1;
    rVelCmdM2 := (rVelFF2 + 0.5 * rCorrPos + rCorrV2) * rUseRatioM2;
    IF ABS(rVelAppl) > 0.001 THEN
        IF rVelAppl > 0.0 THEN
            IF rVelCmdM1 < 0.0 THEN
                rVelCmdM1 := 0.0;
            END_IF;
            IF rVelCmdM2 < 0.0 THEN
                rVelCmdM2 := 0.0;
            END_IF;
        ELSE
            IF rVelCmdM1 > 0.0 THEN
                rVelCmdM1 := 0.0;
            END_IF;
            IF rVelCmdM2 > 0.0 THEN
                rVelCmdM2 := 0.0;
            END_IF;
        END_IF;
    END_IF;
ELSIF (eMode = 2) OR (eMode = 3) THEN
    rTrimFiltered := 0.0;
    IF eMode = 2 THEN
        rVelCmdM1 := ABS(rSpinVel) * rUseRatioM1;
    ELSE
        rVelCmdM1 := -ABS(rSpinVel) * rUseRatioM1;
    END_IF;
    rVelCmdM2 := -rVelCmdM1 * (rUseRatioM2 / rUseRatioM1);
ELSIF eMode = 4 THEN
    (* 0.60 外部直控：两个速度直接来自视觉，不做 trim/sync/斜坡 *)
    rTrimFiltered := 0.0;
    rVelCmdM1 := rVelM1Direct * rUseRatioM1;
    rVelCmdM2 := rVelM2Direct * rUseRatioM2;
ELSE
    rTrimFiltered := 0.0;
    rVelCmdM1 := rVelAppl;
    rVelCmdM2 := rVelAppl;
END_IF;
IF xStop OR NOT xEnable THEN
    rVelCmdM1 := 0.0;
    rVelCmdM2 := 0.0;
END_IF;
IF eMode <> 1 THEN
    xRampLock := FALSE;
ELSIF xRampLock THEN
    IF (ABS(rVelAppl) > 0.001)
            AND (ABS(rVelActM1) >= 0.8 * ABS(rVelAppl))
            AND (ABS(rVelActM2) >= 0.8 * ABS(rVelAppl)) THEN
        xRampLock := FALSE;
    END_IF;
END_IF;
tonRampLock(IN := xRampLock AND (eMode = 1), PT := T#800MS);
IF tonRampLock.Q THEN
    xRampLock := FALSE;
END_IF;
IF (eMode = 1) AND xRampLock THEN
    rVelFbM1 := rVelAppl * rUseRatioM1;
    rVelFbM2 := rVelAppl * rUseRatioM2;
ELSE
    rVelFbM1 := rVelCmdM1;
    rVelFbM2 := rVelCmdM2;
END_IF;
IF (eMode <> 1) OR xStraightEdge THEN
    rVelFbHoldM1 := rVelFbM1;
    rVelFbHoldM2 := rVelFbM2;
ELSE
    IF ABS(rVelFbM1 - rVelFbHoldM1) < 0.004 THEN
        rVelFbM1 := rVelFbHoldM1;
    ELSE
        rVelFbHoldM1 := rVelFbM1;
    END_IF;
    IF ABS(rVelFbM2 - rVelFbHoldM2) < 0.004 THEN
        rVelFbM2 := rVelFbHoldM2;
    ELSE
        rVelFbHoldM2 := rVelFbM2;
    END_IF;
END_IF;

(* ------------------- 7. 双轴 MoveVelocity ------------------- *)
(* 0.54：上升沿锁目标。0.58 每步重触发被 0.59 废除：250Hz 沿风暴反复踢起龙门
   1Hz 共振（现场 acc=0.8：起步快速冲 2 次 ~1s、第三次慢、停死）；两侧 FB/驱动
   接受沿时刻不一致 → M2 漏沿爬速落后（M2 明显慢）。0.59：起步只发一个上升沿，
   一次写入最终目标 + 钳制 Acc/Dec，SM3 自带斜坡 0→目标（0.8 → 0.5s）；
   稳态 trim/sync 更新走限频重触发；减速由 Halt 接管（见第 8 节）。 *)
xHaltBusy := fbHaltM1.Busy OR fbHaltM2.Busy OR fbStopM1.Busy OR fbStopM2.Busy;
IF (eMode = 1) AND xPowerGate AND xPowerSettled AND (ABS(rVelAppl) > 0.001)
        AND NOT xHaltBusy AND NOT xDecelActive AND NOT xDecelDone THEN
    xReqVelM1 := TRUE;
    xReqVelM2 := TRUE;
ELSIF ((eMode = 2) OR (eMode = 3) OR (eMode = 4)) AND xPowerGate AND xPowerSettled AND NOT xHaltBusy
        AND NOT xDecelActive AND NOT xDecelDone THEN
    IF ABS(rVelCmdM1) > 0.001 THEN
        xReqVelM1 := TRUE;
    ELSE
        xReqVelM1 := FALSE;
    END_IF;
    IF ABS(rVelCmdM2) > 0.001 THEN
        xReqVelM2 := TRUE;
    ELSE
        xReqVelM2 := FALSE;
    END_IF;
ELSE
    xReqVelM1 := FALSE;
    xReqVelM2 := FALSE;
END_IF;

xM1Decel := (NOT xReqVelM1) AND xPowerGate AND xMovingM1 AND NOT xStop AND NOT xSoftHold;
xM2Decel := (NOT xReqVelM2) AND xPowerGate AND xMovingM2 AND NOT xStop AND NOT xSoftHold;

(* 方向/换向看 FB 速度（0.54 语义）；减速期由 Halt 接管，无符号穿零 *)
IF ABS(rVelFbM1) > 0.001 THEN
    IF rVelFbM1 >= 0.0 THEN
        eDirM1 := positive;
    ELSE
        eDirM1 := negative;
    END_IF;
END_IF;
IF ABS(rVelFbM2) > 0.001 THEN
    IF rVelFbM2 >= 0.0 THEN
        eDirM2 := positive;
    ELSE
        eDirM2 := negative;
    END_IF;
END_IF;

xDirFlipM1 := xReqVelM1 AND xVelRunPrevM1
              AND (ABS(rVelFbM1) > 0.001) AND (ABS(rVelInPrevM1) > 0.001)
              AND ((rVelFbM1 >= 0.0) <> (rVelInPrevM1 >= 0.0));
xDirFlipM2 := xReqVelM2 AND xVelRunPrevM2
              AND (ABS(rVelFbM2) > 0.001) AND (ABS(rVelInPrevM2) > 0.001)
              AND ((rVelFbM2 >= 0.0) <> (rVelInPrevM2 >= 0.0));
xDirFlipAny := xDirFlipM1 OR xDirFlipM2;

IF (xErrVelM1 OR xErrVelM2) AND NOT xErrVelPrev THEN
    xVelHoldOff := TRUE;
END_IF;
tonVelHold(IN := xVelHoldOff, PT := T#150MS);
IF tonVelHold.Q THEN
    xVelHoldOff := FALSE;
END_IF;
xErrVelPrev := xErrVelM1 OR xErrVelM2;

(* 0.59 提前减速：剩余 ≤ v²/(2·Dec)，v 取双轴实际速度较大者（越保守越早触发）。
   MoveRel 未武装/静止（moved≈0）不触发，短走距不得起步即停。 *)
rDecelDist := 0.0;
IF ABS(rVelActM1) >= ABS(rVelActM2) THEN
    rDecelDist := (ABS(rVelActM1) * ABS(rVelActM1)) / (2.0 * rDecSoft);
ELSE
    rDecelDist := (ABS(rVelActM2) * ABS(rVelActM2)) / (2.0 * rDecSoft);
END_IF;
xMoveRelDecelTrig := xMoveRel AND xArmed AND (NOT xDecelDone)
                     AND (ABS(rMoveDist) > 0.001)
                     AND (ABS(rAvg - rStart) > 0.001)
                     AND (ABS(rAvg - rStart) >= ABS(rMoveDist) - rDecelDist);

(* 松手短窗 Halt 脉冲 + MoveRel 提前减速 Halt 脉冲；减速期禁重复发 *)
xHaltTrig := (xStopping AND (eMode = 0) AND NOT xStop AND NOT xStopFallback
              AND (xMovingM1 OR xMovingM2) AND NOT xDecelActive)
             OR (xMoveRelDecelTrig AND NOT xDecelActive);
(* 0.60 外部直控：任一侧目标为 0 且在动 → 双轴 Halt（停止/失联兜底由 eMode→0 处理） *)
xHaltDemand := xHaltTrig OR ((eMode = 4)
               AND (((NOT xReqVelM1) AND xMovingM1) OR ((NOT xReqVelM2) AND xMovingM2)));
xNeedHaltM1 := xHaltDemand AND NOT xHaltPrev;
xNeedHaltM2 := xNeedHaltM1;
(* 0.56 点动闭锁 + 0.59 减速期撤 Execute（Halt 接管，禁止速度指令抢轴） *)
IF xStop OR NOT xEnable THEN
    xExecHold := FALSE;
ELSIF xDecelActive THEN
    xExecHold := FALSE;
ELSIF xReqVelM1 THEN
    xExecHold := TRUE;
ELSIF (eMode = 0) OR ((eMode = 4) AND (NOT xReqVelM1 OR NOT xReqVelM2)) THEN
    xExecHold := FALSE;
END_IF;
(* 0.59 稳态 trim/sync 更新：限频重触发（≥200ms 一次）。仅非爬坡期（xRampLock 已放）、
   两侧到速、目标与锁存差 ≥0.004。脉冲期撤 Execute 一拍，下一拍上升沿重采样；
   无视觉/同步漂移时永不触发——起步到停车全程一个沿。 *)
xTrimWant := xExecHold AND (NOT xRampLock) AND xVelInVelM1 AND xVelInVelM2
             AND (NOT xDecelActive) AND (NOT xStop)
             AND ((ABS(ABS(rVelFbM1) - rVelLatchM1) >= 0.004)
                  OR (ABS(ABS(rVelFbM2) - rVelLatchM2) >= 0.004));
tonTrimRetrig(IN := xTrimWant, PT := T#200MS);
xTrimPulse := xTrimWant AND tonTrimRetrig.Q AND NOT xTrimPulsePrev;
xTrimPulsePrev := xTrimWant;
(* 0.60 外部直控：目标变化时限频重触发，跟随视觉（无变化不触发，不起沿风暴） *)
xDirectWant := (eMode = 4) AND xExecHold AND (NOT xDecelActive) AND (NOT xStop)
               AND ((ABS(ABS(rVelFbM1) - rVelLatchM1) >= 0.004)
                    OR (ABS(ABS(rVelFbM2) - rVelLatchM2) >= 0.004));
tonDirectRetrig(IN := xDirectWant, PT := tDirectRetrig);
xDirectPulse := xDirectWant AND tonDirectRetrig.Q AND NOT xDirectPulsePrev;
xDirectPulsePrev := xDirectWant;
xExecBoth := NOT xDirFlipAny AND NOT xNeedHaltM1 AND NOT xVelHoldOff AND NOT xTrimPulse
             AND NOT xDirectPulse;
xExecM1 := xExecHold AND xExecBoth;
IF xExecM1 AND NOT xExecPrev THEN
    iVelExecRise := iVelExecRise + 1;
    rVelLatchM1 := ABS(rVelFbM1);
    rVelLatchM2 := ABS(rVelFbM2);
    rAccLatch := rAccSoft;
    rDecLatch := rDecSoft;
ELSIF NOT xExecHold THEN
    rVelLatchM1 := 0.0;
    rVelLatchM2 := 0.0;
END_IF;
fbVelM1(Axis := AxisM1, Execute := xExecM1,
        Velocity := rVelLatchM1, Direction := eDirM1,
        Acceleration := rAccLatch, Deceleration := rDecLatch);
fbVelM2(Axis := AxisM2, Execute := xExecHold AND xExecBoth,
        Velocity := rVelLatchM2, Direction := eDirM2,
        Acceleration := rAccLatch, Deceleration := rDecLatch);

xExecPrev := xExecM1;
xVelRunPrevM1 := xReqVelM1;
xVelRunPrevM2 := xReqVelM2;
rVelInPrevM1 := rVelFbM1;
rVelInPrevM2 := rVelFbM2;

(* ------------------- 8. 停车 ------------------- *)
fbStopM1(Axis := AxisM1, Execute := xStop OR xStopFallback, Deceleration := rDecUse);
fbStopM2(Axis := AxisM2, Execute := xStop OR xStopFallback, Deceleration := rDecUse);
fbHaltM1(Axis := AxisM1, Execute := xNeedHaltM1, Deceleration := rDecSoft);
fbHaltM2(Axis := AxisM2, Execute := xNeedHaltM2, Deceleration := rDecSoft);
xHaltPrev := xHaltDemand;

(* ------------------- 9. 诊断与走距 ------------------- *)
xVelReqM1 := xReqVelM1;
xVelReqM2 := xReqVelM2;
xVelExecM1 := xExecM1;
xVelExecM2 := xExecHold AND xExecBoth;
xVelBusyM1 := fbVelM1.Busy;
xVelBusyM2 := fbVelM2.Busy;
xVelInVelM1 := fbVelM1.InVelocity;
xVelInVelM2 := fbVelM2.InVelocity;
xErrPowerM1 := fbPowerM1.Error;
xErrPowerM2 := fbPowerM2.Error;
xErrVelM1 := fbVelM1.Error;
xErrVelM2 := fbVelM2.Error;
(* 0.60 直控调试输出：实际速度 + 直控在役标志 *)
rVelActM1Out := rVelActM1;
rVelActM2Out := rVelActM2;
xDirectActive := (eMode = 4);

IF xStop OR NOT xEnable OR NOT xMoveRel THEN
    xArmed := FALSE;
    xMoveDone := FALSE;
ELSE
    IF xMoveRel AND NOT xMovePrev THEN
        xArmed := TRUE;
        rStart := rAvg;
    END_IF;
    xMoveDone := xArmed AND (ABS(rAvg - rStart) >= ABS(rMoveDist));
END_IF;
IF NOT xEnable THEN
    iVelExecRise := 0;
END_IF;

(* 0.59 减速状态：松手有速或 MoveRel 提前触发 → Halt 脉冲接管减速；
   双轴静止退出并置到位锁；新点动/旋转/新走距清锁。 *)
IF xMoveRel AND NOT xMovePrev THEN
    xDecelDone := FALSE;
END_IF;
IF xStop OR NOT xEnable THEN
    xDecelActive := FALSE;
    xDecelDone := FALSE;
ELSIF (eMode <> 0) AND (NOT xMoveRel) THEN
    xDecelActive := FALSE;
    xDecelDone := FALSE;
ELSIF xDecelActive THEN
    IF (NOT xMovingM1) AND (NOT xMovingM2) THEN
        xDecelActive := FALSE;
        xDecelDone := TRUE;
    END_IF;
ELSIF (eMode = 0) AND (xMovingM1 OR xMovingM2) THEN
    xDecelActive := TRUE;
ELSIF xMoveRelDecelTrig THEN
    xDecelActive := TRUE;
END_IF;
xMovePrev := xMoveRel;
eModePrev := eMode;
xRegOnPrev := xRegOn;

(* ------------------- 10. M1/M2 驱动诊断慢速 CoE 读取（0.73） ------------------- *)
(* TxPDO 固定映射，诊断对象读不进 PDO；用 ETC_CO_SdoRead 走非循环 SDO。
   100ms 一时隙、24 时隙轮询（单次一个 SDO，一轮约 2.4s）。各自独立缓冲；
   xDone 取 2 字节小端。转矩/电流为‰额定(INT16)，其余原始 UINT16。 *)
tonSdoSlot(IN := NOT tonSdoSlot.Q, PT := T#100MS);
IF tonSdoSlot.Q THEN
    iSdoSlot := iSdoSlot + 1;
    IF iSdoSlot > 23 THEN
        iSdoSlot := 0;
    END_IF;
END_IF;
fbSdoTqM1(xExecute := (iSdoSlot = 0), xAbort := FALSE, usiCom := 1, uiDevice := wSdoDevM1,
    usiChannel := 1, wIndex := 16#6077, bySubindex := 0, udiTimeOut := 500,
    pBuffer := ADR(abyTqM1[0]), szSize := SIZEOF(abyTqM1));
fbSdoCurM1(xExecute := (iSdoSlot = 1), xAbort := FALSE, usiCom := 1, uiDevice := wSdoDevM1,
    usiChannel := 1, wIndex := 16#6078, bySubindex := 0, udiTimeOut := 500,
    pBuffer := ADR(abyCurM1[0]), szSize := SIZEOF(abyCurM1));
fbSdoSwM1(xExecute := (iSdoSlot = 2), xAbort := FALSE, usiCom := 1, uiDevice := wSdoDevM1,
    usiChannel := 1, wIndex := 16#6041, bySubindex := 0, udiTimeOut := 500,
    pBuffer := ADR(abySwM1[0]), szSize := SIZEOF(abySwM1));
fbSdoErrM1(xExecute := (iSdoSlot = 3), xAbort := FALSE, usiCom := 1, uiDevice := wSdoDevM1,
    usiChannel := 1, wIndex := 16#603F, bySubindex := 0, udiTimeOut := 500,
    pBuffer := ADR(abyErrM1[0]), szSize := SIZEOF(abyErrM1));
fbSdoTqMaxM1(xExecute := (iSdoSlot = 4), xAbort := FALSE, usiCom := 1, uiDevice := wSdoDevM1,
    usiChannel := 1, wIndex := 16#6072, bySubindex := 0, udiTimeOut := 500,
    pBuffer := ADR(abyTqMaxM1[0]), szSize := SIZEOF(abyTqMaxM1));
fbSdoLimPM1(xExecute := (iSdoSlot = 5), xAbort := FALSE, usiCom := 1, uiDevice := wSdoDevM1,
    usiChannel := 1, wIndex := 16#60E0, bySubindex := 0, udiTimeOut := 500,
    pBuffer := ADR(abyLimPM1[0]), szSize := SIZEOF(abyLimPM1));
fbSdoLimNM1(xExecute := (iSdoSlot = 6), xAbort := FALSE, usiCom := 1, uiDevice := wSdoDevM1,
    usiChannel := 1, wIndex := 16#60E1, bySubindex := 0, udiTimeOut := 500,
    pBuffer := ADR(abyLimNM1[0]), szSize := SIZEOF(abyLimNM1));
fbSdoModeM1(xExecute := (iSdoSlot = 7), xAbort := FALSE, usiCom := 1, uiDevice := wSdoDevM1,
    usiChannel := 1, wIndex := 16#6060, bySubindex := 0, udiTimeOut := 500,
    pBuffer := ADR(abyModeM1[0]), szSize := SIZEOF(abyModeM1));
fbSdoTq03M1(xExecute := (iSdoSlot = 8), xAbort := FALSE, usiCom := 1, uiDevice := wSdoDevM1,
    usiChannel := 1, wIndex := 16#2403, bySubindex := 0, udiTimeOut := 500,
    pBuffer := ADR(abyTq03M1[0]), szSize := SIZEOF(abyTq03M1));
fbSdoTq04M1(xExecute := (iSdoSlot = 9), xAbort := FALSE, usiCom := 1, uiDevice := wSdoDevM1,
    usiChannel := 1, wIndex := 16#2404, bySubindex := 0, udiTimeOut := 500,
    pBuffer := ADR(abyTq04M1[0]), szSize := SIZEOF(abyTq04M1));
fbSdoTq05M1(xExecute := (iSdoSlot = 10), xAbort := FALSE, usiCom := 1, uiDevice := wSdoDevM1,
    usiChannel := 1, wIndex := 16#2405, bySubindex := 0, udiTimeOut := 500,
    pBuffer := ADR(abyTq05M1[0]), szSize := SIZEOF(abyTq05M1));
fbSdoTq06M1(xExecute := (iSdoSlot = 11), xAbort := FALSE, usiCom := 1, uiDevice := wSdoDevM1,
    usiChannel := 1, wIndex := 16#2406, bySubindex := 0, udiTimeOut := 500,
    pBuffer := ADR(abyTq06M1[0]), szSize := SIZEOF(abyTq06M1));
fbSdoTqM2(xExecute := (iSdoSlot = 12), xAbort := FALSE, usiCom := 1, uiDevice := wSdoDevM2,
    usiChannel := 1, wIndex := 16#6077, bySubindex := 0, udiTimeOut := 500,
    pBuffer := ADR(abyTqM2[0]), szSize := SIZEOF(abyTqM2));
fbSdoCurM2(xExecute := (iSdoSlot = 13), xAbort := FALSE, usiCom := 1, uiDevice := wSdoDevM2,
    usiChannel := 1, wIndex := 16#6078, bySubindex := 0, udiTimeOut := 500,
    pBuffer := ADR(abyCurM2[0]), szSize := SIZEOF(abyCurM2));
fbSdoSwM2(xExecute := (iSdoSlot = 14), xAbort := FALSE, usiCom := 1, uiDevice := wSdoDevM2,
    usiChannel := 1, wIndex := 16#6041, bySubindex := 0, udiTimeOut := 500,
    pBuffer := ADR(abySwM2[0]), szSize := SIZEOF(abySwM2));
fbSdoErrM2(xExecute := (iSdoSlot = 15), xAbort := FALSE, usiCom := 1, uiDevice := wSdoDevM2,
    usiChannel := 1, wIndex := 16#603F, bySubindex := 0, udiTimeOut := 500,
    pBuffer := ADR(abyErrM2[0]), szSize := SIZEOF(abyErrM2));
fbSdoTqMaxM2(xExecute := (iSdoSlot = 16), xAbort := FALSE, usiCom := 1, uiDevice := wSdoDevM2,
    usiChannel := 1, wIndex := 16#6072, bySubindex := 0, udiTimeOut := 500,
    pBuffer := ADR(abyTqMaxM2[0]), szSize := SIZEOF(abyTqMaxM2));
fbSdoLimPM2(xExecute := (iSdoSlot = 17), xAbort := FALSE, usiCom := 1, uiDevice := wSdoDevM2,
    usiChannel := 1, wIndex := 16#60E0, bySubindex := 0, udiTimeOut := 500,
    pBuffer := ADR(abyLimPM2[0]), szSize := SIZEOF(abyLimPM2));
fbSdoLimNM2(xExecute := (iSdoSlot = 18), xAbort := FALSE, usiCom := 1, uiDevice := wSdoDevM2,
    usiChannel := 1, wIndex := 16#60E1, bySubindex := 0, udiTimeOut := 500,
    pBuffer := ADR(abyLimNM2[0]), szSize := SIZEOF(abyLimNM2));
fbSdoModeM2(xExecute := (iSdoSlot = 19), xAbort := FALSE, usiCom := 1, uiDevice := wSdoDevM2,
    usiChannel := 1, wIndex := 16#6060, bySubindex := 0, udiTimeOut := 500,
    pBuffer := ADR(abyModeM2[0]), szSize := SIZEOF(abyModeM2));
fbSdoTq03M2(xExecute := (iSdoSlot = 20), xAbort := FALSE, usiCom := 1, uiDevice := wSdoDevM2,
    usiChannel := 1, wIndex := 16#2403, bySubindex := 0, udiTimeOut := 500,
    pBuffer := ADR(abyTq03M2[0]), szSize := SIZEOF(abyTq03M2));
fbSdoTq04M2(xExecute := (iSdoSlot = 21), xAbort := FALSE, usiCom := 1, uiDevice := wSdoDevM2,
    usiChannel := 1, wIndex := 16#2404, bySubindex := 0, udiTimeOut := 500,
    pBuffer := ADR(abyTq04M2[0]), szSize := SIZEOF(abyTq04M2));
fbSdoTq05M2(xExecute := (iSdoSlot = 22), xAbort := FALSE, usiCom := 1, uiDevice := wSdoDevM2,
    usiChannel := 1, wIndex := 16#2405, bySubindex := 0, udiTimeOut := 500,
    pBuffer := ADR(abyTq05M2[0]), szSize := SIZEOF(abyTq05M2));
fbSdoTq06M2(xExecute := (iSdoSlot = 23), xAbort := FALSE, usiCom := 1, uiDevice := wSdoDevM2,
    usiChannel := 1, wIndex := 16#2406, bySubindex := 0, udiTimeOut := 500,
    pBuffer := ADR(abyTq06M2[0]), szSize := SIZEOF(abyTq06M2));
IF fbSdoTqM1.xDone THEN
    wSdoRaw := BYTE_TO_WORD(abyTqM1[0]) OR SHL(BYTE_TO_WORD(abyTqM1[1]), 8);
    rTorqueActM1 := INT_TO_REAL(WORD_TO_INT(wSdoRaw));
END_IF;
IF fbSdoCurM1.xDone THEN
    wSdoRaw := BYTE_TO_WORD(abyCurM1[0]) OR SHL(BYTE_TO_WORD(abyCurM1[1]), 8);
    rCurrentActM1 := INT_TO_REAL(WORD_TO_INT(wSdoRaw));
END_IF;
IF fbSdoSwM1.xDone THEN
    wSwM1 := BYTE_TO_WORD(abySwM1[0]) OR SHL(BYTE_TO_WORD(abySwM1[1]), 8);
END_IF;
IF fbSdoErrM1.xDone THEN
    wErrM1 := BYTE_TO_WORD(abyErrM1[0]) OR SHL(BYTE_TO_WORD(abyErrM1[1]), 8);
END_IF;
IF fbSdoTqMaxM1.xDone THEN
    wTqMaxM1 := BYTE_TO_WORD(abyTqMaxM1[0]) OR SHL(BYTE_TO_WORD(abyTqMaxM1[1]), 8);
END_IF;
IF fbSdoLimPM1.xDone THEN
    wLimPM1 := BYTE_TO_WORD(abyLimPM1[0]) OR SHL(BYTE_TO_WORD(abyLimPM1[1]), 8);
END_IF;
IF fbSdoLimNM1.xDone THEN
    wLimNM1 := BYTE_TO_WORD(abyLimNM1[0]) OR SHL(BYTE_TO_WORD(abyLimNM1[1]), 8);
END_IF;
IF fbSdoModeM1.xDone THEN
    wModeM1 := BYTE_TO_WORD(abyModeM1[0]) OR SHL(BYTE_TO_WORD(abyModeM1[1]), 8);
END_IF;
IF fbSdoTq03M1.xDone THEN
    wTq03M1 := BYTE_TO_WORD(abyTq03M1[0]) OR SHL(BYTE_TO_WORD(abyTq03M1[1]), 8);
END_IF;
IF fbSdoTq04M1.xDone THEN
    wTq04M1 := BYTE_TO_WORD(abyTq04M1[0]) OR SHL(BYTE_TO_WORD(abyTq04M1[1]), 8);
END_IF;
IF fbSdoTq05M1.xDone THEN
    wTq05M1 := BYTE_TO_WORD(abyTq05M1[0]) OR SHL(BYTE_TO_WORD(abyTq05M1[1]), 8);
END_IF;
IF fbSdoTq06M1.xDone THEN
    wTq06M1 := BYTE_TO_WORD(abyTq06M1[0]) OR SHL(BYTE_TO_WORD(abyTq06M1[1]), 8);
END_IF;
IF fbSdoTqM2.xDone THEN
    wSdoRaw := BYTE_TO_WORD(abyTqM2[0]) OR SHL(BYTE_TO_WORD(abyTqM2[1]), 8);
    rTorqueActM2 := INT_TO_REAL(WORD_TO_INT(wSdoRaw));
END_IF;
IF fbSdoCurM2.xDone THEN
    wSdoRaw := BYTE_TO_WORD(abyCurM2[0]) OR SHL(BYTE_TO_WORD(abyCurM2[1]), 8);
    rCurrentActM2 := INT_TO_REAL(WORD_TO_INT(wSdoRaw));
END_IF;
IF fbSdoSwM2.xDone THEN
    wSwM2 := BYTE_TO_WORD(abySwM2[0]) OR SHL(BYTE_TO_WORD(abySwM2[1]), 8);
END_IF;
IF fbSdoErrM2.xDone THEN
    wErrM2 := BYTE_TO_WORD(abyErrM2[0]) OR SHL(BYTE_TO_WORD(abyErrM2[1]), 8);
END_IF;
IF fbSdoTqMaxM2.xDone THEN
    wTqMaxM2 := BYTE_TO_WORD(abyTqMaxM2[0]) OR SHL(BYTE_TO_WORD(abyTqMaxM2[1]), 8);
END_IF;
IF fbSdoLimPM2.xDone THEN
    wLimPM2 := BYTE_TO_WORD(abyLimPM2[0]) OR SHL(BYTE_TO_WORD(abyLimPM2[1]), 8);
END_IF;
IF fbSdoLimNM2.xDone THEN
    wLimNM2 := BYTE_TO_WORD(abyLimNM2[0]) OR SHL(BYTE_TO_WORD(abyLimNM2[1]), 8);
END_IF;
IF fbSdoModeM2.xDone THEN
    wModeM2 := BYTE_TO_WORD(abyModeM2[0]) OR SHL(BYTE_TO_WORD(abyModeM2[1]), 8);
END_IF;
IF fbSdoTq03M2.xDone THEN

(* ------------------- 11. 强制 X 双驱 CSV 速度模式（0.77） ------------------- *)
(* SMC_SetControllerMode 切换最长约 1000 周期(~4s)：必须保持 bExecute 到 Done/Error。
   0.76 每秒脉冲会在切完前重启 -> 永远完不成(w74 恒 0)。这里空闲且使能时切一次并保持。 *)
IF NOT xEnable OR xStop THEN
    xModeVelDoneM1 := FALSE;
    xModeVelDoneM2 := FALSE;
END_IF;
xModeReqM1 := xForceCsv AND xEnable AND NOT xStop AND NOT xStopping AND NOT xDecelActive
              AND (eMode = 0) AND NOT xModeVelDoneM1;
fbSetModeM1(Axis := AxisM1, bExecute := xModeReqM1, nControllerMode := SMC_velocity);
IF fbSetModeM1.bDone OR fbSetModeM1.bError THEN
    xModeVelDoneM1 := TRUE;
END_IF;
xModeCsvM1 := fbSetModeM1.bDone OR (WORD_TO_INT(wModeM1) = 9);
xModeCsvErrM1 := fbSetModeM1.bError;
xModeReqM2 := xForceCsv AND xEnable AND NOT xStop AND NOT xStopping AND NOT xDecelActive
              AND (eMode = 0) AND NOT xModeVelDoneM2;
fbSetModeM2(Axis := AxisM2, bExecute := xModeReqM2, nControllerMode := SMC_velocity);
IF fbSetModeM2.bDone OR fbSetModeM2.bError THEN
    xModeVelDoneM2 := TRUE;
END_IF;
xModeCsvM2 := fbSetModeM2.bDone OR (WORD_TO_INT(wModeM2) = 9);
xModeCsvErrM2 := fbSetModeM2.bError;

    wTq03M2 := BYTE_TO_WORD(abyTq03M2[0]) OR SHL(BYTE_TO_WORD(abyTq03M2[1]), 8);
END_IF;
IF fbSdoTq04M2.xDone THEN
    wTq04M2 := BYTE_TO_WORD(abyTq04M2[0]) OR SHL(BYTE_TO_WORD(abyTq04M2[1]), 8);
END_IF;
IF fbSdoTq05M2.xDone THEN
    wTq05M2 := BYTE_TO_WORD(abyTq05M2[0]) OR SHL(BYTE_TO_WORD(abyTq05M2[1]), 8);
END_IF;
IF fbSdoTq06M2.xDone THEN
    wTq06M2 := BYTE_TO_WORD(abyTq06M2[0]) OR SHL(BYTE_TO_WORD(abyTq06M2[1]), 8);
END_IF;
xParamErr := fbSdoTqM1.xError OR fbSdoCurM1.xError OR fbSdoSwM1.xError OR fbSdoErrM1.xError OR fbSdoTqMaxM1.xError OR fbSdoLimPM1.xError OR fbSdoLimNM1.xError OR fbSdoModeM1.xError OR fbSdoTq03M1.xError OR fbSdoTq04M1.xError OR fbSdoTq05M1.xError OR fbSdoTq06M1.xError OR fbSdoTqM2.xError OR fbSdoCurM2.xError OR fbSdoSwM2.xError OR fbSdoErrM2.xError OR fbSdoTqMaxM2.xError OR fbSdoLimPM2.xError OR fbSdoLimNM2.xError OR fbSdoModeM2.xError OR fbSdoTq03M2.xError OR fbSdoTq04M2.xError OR fbSdoTq05M2.xError OR fbSdoTq06M2.xError;

(* ------------------- 12. 启动直写 0x6060=9(CSV) 再运动（0.75） ------------------- *)
(* 若 0.74 的 SMC_SetControllerMode 被驱动/PDO 拒绝，用 ETC_CO_SdoWrite4 直写 0x6060=9。
   空闲且使能时写一次；Done/Error 都锁，避免反复。 *)
IF NOT xEnable OR xStop THEN
    xModeWrDoneM1 := FALSE;
    xModeWrDoneM2 := FALSE;
END_IF;
abyModeWr[1] := 9;
fbWrModeM1(xExecute := xForceCsv AND xEnable AND NOT xStop AND NOT xDecelActive
                        AND (eMode = 0) AND NOT xModeWrDoneM1,
    xAbort := FALSE, usiCom := 1, uiDevice := wSdoDevM1, usiChannel := 1,
    wIndex := 16#6060, bySubindex := 0, udiTimeOut := 500,
    abyData := abyModeWr, usiDataLength := 1);
IF fbWrModeM1.xDone OR fbWrModeM1.xError THEN
    xModeWrDoneM1 := TRUE;
END_IF;
xModeWrErrM1 := fbWrModeM1.xError;
fbWrModeM2(xExecute := xForceCsv AND xEnable AND NOT xStop AND NOT xDecelActive
                        AND (eMode = 0) AND NOT xModeWrDoneM2,
    xAbort := FALSE, usiCom := 1, uiDevice := wSdoDevM2, usiChannel := 1,
    wIndex := 16#6060, bySubindex := 0, udiTimeOut := 500,
    abyData := abyModeWr, usiDataLength := 1);
IF fbWrModeM2.xDone OR fbWrModeM2.xError THEN
    xModeWrDoneM2 := TRUE;
END_IF;
xModeWrErrM2 := fbWrModeM2.xError;
          
END_FUNCTION_BLOCK

PROGRAM PRG_Logic
  VAR
    tonHold : TON;
    tonReady : TON;
    xResetPulse : BOOL;
    xResetPrev : BOOL;
    xSafe : BOOL;
    xAutoStartPrev : BOOL;
    xAutoStartEdge : BOOL;
    rRHold : REAL;
    iPass : INT;
    xAutoTareSent : BOOL;
    xHomeTrigY : BOOL;
    xHomeTrigZ : BOOL;
    xHomeTrigR : BOOL;
    xHomeTrigYPrev : BOOL;
    xHomeTrigZPrev : BOOL;
    xHomeTrigRPrev : BOOL;
    xAnyHomeBusy : BOOL;
    xReadyAll : BOOL;
    xPanelSrc : BOOL;  (* eCtrlSrc=0：面板/触摸屏源 *)
    xJogXPosM : BOOL;  (* 合并后点动（HMI/Web OR 面板键） *)
    xJogXNegM : BOOL;
    xJogYPosM : BOOL;
    xJogYNegM : BOOL;
    xJogZPosM : BOOL;
    xJogZNegM : BOOL;
    xJogRPosM : BOOL;
    xJogRNegM : BOOL;
    xCmdJogXPos : BOOL;
    xCmdJogXNeg : BOOL;
    xCmdSpinL : BOOL;
    xCmdSpinR : BOOL;
    xCmdJogYPos : BOOL;
    xCmdJogYNeg : BOOL;
    xCmdJogZPos : BOOL;
    xCmdJogZNeg : BOOL;
    xCmdJogRPos : BOOL;
    xCmdJogRNeg : BOOL;
    xCmdForceFollow : BOOL;
    xCmdMoveRelX : BOOL;
    xCmdMoveRelY : BOOL;
    xCmdMoveAbsY : BOOL;
    xCmdHoldR : BOOL;
    tonDirectWd : TON;
    xVisSeen : BOOL;
    xVisReq : BOOL;
    xDirectSafe : BOOL;
    Vis_wSeqPrev : WORD;
    rVelM1Sel : REAL;
    rVelM2Sel : REAL;
    tonDirect2 : TON;
    xDirectSeen : BOOL;
    wDirectSeqPrev : WORD;
    xDirect2Enable : BOOL;
    xHmiDirectVelX : BOOL;
    xDirectVelY : BOOL;
    xDirectVelZ : BOOL;
    xDirectVelR : BOOL;
    xDirectAbsY : BOOL;
    xDirectAbsZ : BOOL;
    xDirectAbsR : BOOL;
    xDirectRelY : BOOL;
    xDirectRelZ : BOOL;
    xDirectRelR : BOOL;
    rDirectFeedY : REAL;
    rDirectFeedZ : REAL;
    rDirectFeedR : REAL;
    rDirectVelYSel : REAL;
    rDirectVelZSel : REAL;
    rDirectVelRSel : REAL;
    rDirectPosYSel : REAL;
    rDirectPosZSel : REAL;
    rDirectPosRSel : REAL;
  END_VAR

            (* PRG_Logic — 消费已仲裁 HMI_* + 面板键；写 AxisCmd_*；状态只读派生（无状态机耦合）。
   禁止 CALL Axis / FB_Servo。 *)

(* ===== 急停锁存 / 长按复位 ===== *)
IF NOT HMI_xEStop THEN
    xEStopLatched := TRUE;
END_IF;
tonHold(IN := HMI_xStop AND HMI_xEStop, PT := T#3S);
xResetPulse := (HMI_xStopHold3s OR tonHold.Q) AND NOT xResetPrev;
xResetPrev := HMI_xStopHold3s OR tonHold.Q;
IF xResetPulse THEN
    xEStopLatched := FALSE;
    AxisCmd_xResetFault := TRUE;
    iAutoStep := 0;
    iPass := 0;
    Force_xSlaveFail := FALSE;
ELSE
    AxisCmd_xResetFault := FALSE;
END_IF;

(* 故障汇总：各轴 Errorstop（同步跳闸已废，不再 OR AxisFb_xSyncFault） *)
xFaultAggregate := AxisFb_xFaultM1 OR AxisFb_xFaultM2 OR AxisFb_xFaultY OR AxisFb_xFaultZ
    OR (xM5Ready AND AxisFb_xFaultR);

IF HMI_xAutoMode THEN eOpMode := 1; ELSE eOpMode := 0; END_IF;
HMI_eOpMode := eOpMode;

(* 安全 / 使能 —— 去耦：只看急停 + 故障 *)
xSafe := HMI_xEStop AND NOT xEStopLatched;
AxisCmd_xPower := xSafe;
AxisCmd_xStopAll := HMI_xStop OR NOT xSafe OR xFaultAggregate OR HMI_xAutoAbort;

(* ===== 0.68 全轴直控：心跳看门狗 + 安全门（视觉与操作员共用） ===== *)
(* HMI_wDirectSeq 300ms 不变 -> 心跳丢失，退出直控并停 *)
IF HMI_wDirectSeq <> wDirectSeqPrev THEN
    wDirectSeqPrev := HMI_wDirectSeq;
    xDirectSeen := TRUE;
    tonDirect2(IN := FALSE);
    tonDirect2(IN := TRUE, PT := Cfg_tDirectTimeout);
END_IF;
tonDirect2();
Direct2_xOnline := xDirectSeen AND NOT tonDirect2.Q;
Direct2_wSeqEcho := HMI_wDirectSeq;
(* 直控安全门：手动模式 + 安全 + 未停止 + 无轴故障 *)
Direct2_xSafe := xSafe AND (eOpMode = 0) AND NOT HMI_xStop AND NOT xFaultAggregate;
xDirect2Enable := HMI_xDirectEnable AND Direct2_xOnline AND Direct2_xSafe;

(* ===== 0.60/0.68 X 视觉/Web 直控：视觉(Vis_*)
(* 视觉心跳：Vis_wSeq 变化则复位看门狗；200ms 无变化 -> 离线 *)
IF Vis_wSeq <> Vis_wSeqPrev THEN
    Vis_wSeqPrev := Vis_wSeq;
    xVisSeen := TRUE;
    tonDirectWd(IN := FALSE);
    tonDirectWd(IN := TRUE, PT := T#200MS);
END_IF;
tonDirectWd();
Direct_xOnline := xVisSeen AND NOT tonDirectWd.Q;
Direct_wSeqEcho := Vis_wSeq;

xVisReq := Vis_xEnable AND Direct_xOnline;
xDirectSafe := Direct2_xSafe;
xHmiDirectVelX := HMI_xDirectEnable AND (HMI_iDirectModeX = UINT#1) AND Direct2_xOnline;
IF xVisReq THEN
    rVelM1Sel := Vis_rVelM1Set;
    rVelM2Sel := Vis_rVelM2Set;
ELSIF xHmiDirectVelX THEN
    rVelM1Sel := LIMIT(-Cfg_rDirectVelMaxX, HMI_rVelM1Set, Cfg_rDirectVelMaxX);
    rVelM2Sel := LIMIT(-Cfg_rDirectVelMaxX, HMI_rVelM2Set, Cfg_rDirectVelMaxX);
ELSE
    rVelM1Sel := 0.0;
    rVelM2Sel := 0.0;
END_IF;

Direct_xEnable := (xVisReq OR xHmiDirectVelX) AND xDirectSafe;
AxisCmd_xDirectVel := Direct_xEnable;
AxisCmd_rVelM1Set := rVelM1Sel;
AxisCmd_rVelM2Set := rVelM2Sel;
Direct2_xActiveX := Direct_xEnable;

(* ===== 0.68 Y/Z/R 直控：0=idle(减速停) 1=速度 2=绝对 3=相对 ===== *)
(* 先清本地指令，模式仲裁后扫描末尾一次性写 AxisCmd_*，避免同扫描 TRUE->FALSE 空窗 *)
xDirectVelY := FALSE; xDirectVelZ := FALSE; xDirectVelR := FALSE;
xDirectAbsY := FALSE; xDirectAbsZ := FALSE; xDirectAbsR := FALSE;
xDirectRelY := FALSE; xDirectRelZ := FALSE; xDirectRelR := FALSE;
rDirectVelYSel := 0.0; rDirectVelZSel := 0.0; rDirectVelRSel := 0.0;
rDirectPosYSel := 0.0; rDirectPosZSel := 0.0; rDirectPosRSel := 0.0;
(* 限幅后的进给速度；模式 2/3 用同一进给速度，避免位置模式下速度=0 *)
rDirectFeedY := LIMIT(0.0, ABS(HMI_rDirectVelY), Cfg_rDirectVelMaxY);
IF rDirectFeedY < 1.0E-4 THEN rDirectFeedY := Cfg_rDirectVelMaxY; END_IF;
rDirectFeedZ := LIMIT(0.0, ABS(HMI_rDirectVelZ), Cfg_rDirectVelMaxZ);
IF rDirectFeedZ < 1.0E-4 THEN rDirectFeedZ := Cfg_rDirectVelMaxZ; END_IF;
rDirectFeedR := LIMIT(0.0, ABS(HMI_rDirectVelR), Cfg_rDirectVelMaxR);
IF rDirectFeedR < 1.0E-4 THEN rDirectFeedR := Cfg_rDirectVelMaxR; END_IF;

IF xDirect2Enable THEN
    CASE HMI_iDirectModeY OF
        1:
            xDirectVelY := TRUE;
            rDirectVelYSel := LIMIT(-Cfg_rDirectVelMaxY, HMI_rDirectVelY, Cfg_rDirectVelMaxY);
        2:
            xDirectAbsY := TRUE;
            rDirectPosYSel := LIMIT(Cfg_rLimYNeg, HMI_rDirectPosY, Cfg_rLimYPos);
            rDirectVelYSel := rDirectFeedY;
        3:
            xDirectRelY := TRUE;
            rDirectPosYSel := HMI_rDirectPosY;
            rDirectVelYSel := rDirectFeedY;
    END_CASE;
    CASE HMI_iDirectModeZ OF
        1:
            xDirectVelZ := TRUE;
            rDirectVelZSel := LIMIT(-Cfg_rDirectVelMaxZ, HMI_rDirectVelZ, Cfg_rDirectVelMaxZ);
        2:
            xDirectAbsZ := TRUE;
            rDirectPosZSel := LIMIT(Cfg_rLimZNeg, HMI_rDirectPosZ, Cfg_rLimZPos);
            rDirectVelZSel := rDirectFeedZ;
        3:
            xDirectRelZ := TRUE;
            rDirectPosZSel := HMI_rDirectPosZ;
            rDirectVelZSel := rDirectFeedZ;
    END_CASE;
    CASE HMI_iDirectModeR OF
        1:
            xDirectVelR := TRUE;
            rDirectVelRSel := LIMIT(-Cfg_rDirectVelMaxR, HMI_rDirectVelR, Cfg_rDirectVelMaxR);
        2:
            xDirectAbsR := TRUE;
            rDirectPosRSel := LIMIT(Cfg_rLimRNeg, HMI_rDirectPosR, Cfg_rLimRPos);
            rDirectVelRSel := rDirectFeedR;
        3:
            xDirectRelR := TRUE;
            rDirectPosRSel := HMI_rDirectPosR;
            rDirectVelRSel := rDirectFeedR;
    END_CASE;
END_IF;
Direct2_xActiveY := xDirect2Enable AND (HMI_iDirectModeY <> UINT#0);
Direct2_xActiveZ := xDirect2Enable AND (HMI_iDirectModeZ <> UINT#0);
Direct2_xActiveR := xDirect2Enable AND (HMI_iDirectModeR <> UINT#0);

(* 力/纠偏参数下发 *)
rForceKp := HMI_rKpForce;
IF rForceKp < 1.0E-6 THEN rForceKp := 1.0; END_IF;
AxisCmd_rForceSet := HMI_rForceSet;
AxisCmd_rForceKp := rForceKp;
AxisCmd_rForceVelMax := ABS(HMI_rAutoVelZ);
IF AxisCmd_rForceVelMax < 1.0E-6 THEN AxisCmd_rForceVelMax := ABS(HMI_rJogVelZ); END_IF;
AxisCmd_rHeadingErr := HMI_rHeadingErr;

IF HMI_xForceSimEnable THEN
    rForceAct := HMI_rForceSim;
END_IF;
HMI_rForceShow := rForceAct;
HMI_rForceSetEcho := HMI_rForceSet;
(* 力峰值（绝对值）+ 原始计数：复位脉冲先清零，再对新值取峰值 *)
IF HMI_xForcePeakReset THEN Force_rPeak := 0.0; END_IF;
Force_rPeak := MAX(Force_rPeak, ABS(HMI_rForceShow));
Force_wRaw := Force_wInRaw;

AxisCmd_rJogVelX := HMI_rJogVelX;
AxisCmd_rSpinVel := HMI_rSpinVel;
AxisCmd_rJogVelY := HMI_rJogVelY;
AxisCmd_rJogVelZ := HMI_rJogVelZ;
AxisCmd_rJogVelR := HMI_rJogVelR;
AxisCmd_rWheelBase := LIMIT(4.0, HMI_rWheelBase, 6.0);
(* 每轴加减速：仅未填(≈0)才兜底 100。X 已调到与点动速度同量级时必须原样下发。 *)
AxisCmd_rAccX := HMI_rAccX; IF AxisCmd_rAccX < 0.05 THEN AxisCmd_rAccX := 100.0; END_IF;
AxisCmd_rDecX := HMI_rDecX; IF AxisCmd_rDecX < 0.05 THEN AxisCmd_rDecX := 100.0; END_IF;
AxisCmd_rAccY := HMI_rAccY; IF AxisCmd_rAccY < 1.0 THEN AxisCmd_rAccY := 100.0; END_IF;
AxisCmd_rDecY := HMI_rDecY; IF AxisCmd_rDecY < 1.0 THEN AxisCmd_rDecY := 100.0; END_IF;
AxisCmd_rAccZ := HMI_rAccZ; IF AxisCmd_rAccZ < 1.0 THEN AxisCmd_rAccZ := 100.0; END_IF;
AxisCmd_rDecZ := HMI_rDecZ; IF AxisCmd_rDecZ < 1.0 THEN AxisCmd_rDecZ := 100.0; END_IF;
AxisCmd_rAccR := HMI_rAccR; IF AxisCmd_rAccR < 1.0 THEN AxisCmd_rAccR := 100.0; END_IF;
AxisCmd_rDecR := HMI_rDecR; IF AxisCmd_rDecR < 1.0 THEN AxisCmd_rDecR := 100.0; END_IF;

(* 限位联锁：物理限位输入 ∨ 可配置硬限位（Cfg_rLim*，FB_Servo 内另有最终闸门） *)
xIlk_BlockYPlus := I_xLimYPos OR (AxisFb_rPosY >= Cfg_rLimYPos);
xIlk_BlockYNeg := I_xLimYNeg OR (AxisFb_rPosY <= Cfg_rLimYNeg);
xIlk_BlockZPlus := I_xLimZPos OR (AxisFb_rPosZ >= Cfg_rLimZPos);
xIlk_BlockZNeg := I_xLimZNeg OR (AxisFb_rPosZ <= Cfg_rLimZNeg);

(* 运动位先写入局部，扫描结束一次性交给 AxisCmd。
   禁止先清 GVL 再置位：ETHERCAT 优先级更高，会采到 FALSE 空窗，点动 Acc 被重爬三次。 *)
xCmdJogXPos := FALSE; xCmdJogXNeg := FALSE;
xCmdSpinL := FALSE; xCmdSpinR := FALSE;
xCmdJogYPos := FALSE; xCmdJogYNeg := FALSE;
xCmdJogZPos := FALSE; xCmdJogZNeg := FALSE;
xCmdJogRPos := FALSE; xCmdJogRNeg := FALSE;
xCmdForceFollow := FALSE;
xCmdMoveRelX := FALSE;
xCmdMoveRelY := FALSE;
xCmdMoveAbsY := FALSE;
xCmdHoldR := FALSE;
(* 视觉差速：手动点动与自动走距都下发 Kp；FB 仅在直行模式用 *)
AxisCmd_rTrackKp := HMI_rKpTrack;
Logic_xForceTare := FALSE;

xAutoStartEdge := HMI_xAutoStart AND NOT xAutoStartPrev;
xAutoStartPrev := HMI_xAutoStart;

IF HMI_xAutoAbort OR NOT xSafe OR xFaultAggregate THEN
    iAutoStep := 0;
    iPass := 0;
    HMI_xAutoBusy := FALSE;
END_IF;

(* ===== 点动源合并：面板键（仅面板/触摸屏源时）OR 触摸屏/Web ===== *)
xPanelSrc := (eCtrlSrc = 0);
xJogXPosM := HMI_xJogXPos OR (xPanelSrc AND JogFwd);
xJogXNegM := HMI_xJogXNeg OR (xPanelSrc AND JogBwd);
xJogYPosM := HMI_xJogYPos OR (xPanelSrc AND JogRight);
xJogYNegM := HMI_xJogYNeg OR (xPanelSrc AND JogLeft);
xJogZPosM := HMI_xJogZPos OR (xPanelSrc AND JogUp);
xJogZNegM := HMI_xJogZNeg OR (xPanelSrc AND JogDown);
xJogRPosM := HMI_xJogRPos OR (xPanelSrc AND JogClockAdd);
xJogRNegM := HMI_xJogRNeg OR (xPanelSrc AND JogClockMis);

(* ===== 手动 ===== *)
IF xSafe AND (eOpMode = 0) AND NOT HMI_xStop AND NOT xFaultAggregate THEN
    (* 直控在役时屏蔽 X 手动（旋转/点动），速度由视觉/Web 直控通道给 *)
    IF (HMI_xSpinLeft XOR HMI_xSpinRight) AND NOT Direct_xEnable THEN
        xCmdSpinL := HMI_xSpinLeft;
        xCmdSpinR := HMI_xSpinRight;
    ELSIF (xJogXPosM XOR xJogXNegM) AND NOT Direct_xEnable THEN
        xCmdJogXPos := xJogXPosM;
        xCmdJogXNeg := xJogXNegM;
    END_IF;
    xCmdJogYPos := xJogYPosM AND NOT xIlk_BlockYPlus AND NOT xDirect2Enable;
    xCmdJogYNeg := xJogYNegM AND NOT xIlk_BlockYNeg AND NOT xDirect2Enable;
    IF HMI_xForceGuide AND NOT xDirect2Enable THEN
        xCmdForceFollow := TRUE;
    ELSE
        xCmdJogZPos := xJogZPosM AND NOT xIlk_BlockZPlus AND NOT xDirect2Enable;
        xCmdJogZNeg := xJogZNegM AND NOT xIlk_BlockZNeg AND NOT xDirect2Enable;
    END_IF;
    IF xM5Ready AND NOT xDirect2Enable THEN
        xCmdJogRPos := xJogRPosM;
        xCmdJogRNeg := xJogRNegM;
    END_IF;
END_IF;

(* ===== 自动多道循环 ===== *)
IF xSafe AND (eOpMode = 1) AND NOT HMI_xStop AND NOT xFaultAggregate THEN
    IF iAutoStep = 0 AND xAutoStartEdge THEN
        rRHold := AxisFb_rPosR;
        xAutoTareSent := FALSE;
        HMI_xAutoDone := FALSE;
        HMI_xAutoBusy := TRUE;
        iPass := 1;
        iAutoStep := 1;
    END_IF;

    CASE iAutoStep OF
        1:
            xCmdHoldR := TRUE;
            AxisCmd_rRHoldPos := rRHold;
            AxisCmd_rTrackKp := HMI_rKpTrack;
            AxisCmd_rMoveDistX := HMI_rAutoDistX;
            AxisCmd_rMoveVelX := HMI_rAutoVelX;
            xCmdMoveRelX := TRUE;
            IF AxisFb_xMoveDoneX THEN
                xCmdMoveRelX := FALSE;
                iAutoStep := 2;
            END_IF;
        2:
            xCmdHoldR := TRUE;
            AxisCmd_rRHoldPos := rRHold;
            AxisCmd_rMoveAbsPosY := 0.0;
            AxisCmd_rMoveVelY := HMI_rAutoVelY;
            xCmdMoveAbsY := TRUE;
            IF AxisFb_xStandstillY AND (ABS(AxisFb_rPosY) < 0.005) THEN
                xCmdMoveAbsY := FALSE;
                xAutoTareSent := FALSE;
                iAutoStep := 3;
            END_IF;
        3:
            xCmdHoldR := TRUE;
            AxisCmd_rRHoldPos := rRHold;
            IF NOT xAutoTareSent THEN
                Logic_xForceTare := TRUE;
                xAutoTareSent := TRUE;
            END_IF;
            xCmdForceFollow := TRUE;
            IF rForceAct >= HMI_rForceSet THEN
                iAutoStep := 4;
            END_IF;
        4:
            xCmdHoldR := TRUE;
            AxisCmd_rRHoldPos := rRHold;
            xCmdForceFollow := TRUE;
            AxisCmd_rMoveDistY := AxisCmd_rWheelBase;
            AxisCmd_rMoveVelY := HMI_rAutoVelY;
            xCmdMoveRelY := TRUE;
            IF AxisFb_xMoveDoneY THEN
                xCmdMoveRelY := FALSE;
                iAutoStep := 5;
            END_IF;
        5:
            IF iPass < HMI_iAutoPasses THEN
                iPass := iPass + 1;
                iAutoStep := 1;
            ELSE
                iAutoStep := 6;
            END_IF;
        6:
            HMI_xAutoBusy := FALSE;
            HMI_xAutoDone := TRUE;
            iAutoStep := 0;
            iPass := 0;
    END_CASE;
END_IF;

(* ===== 回零：Y/Z/R；同时只回一轴 ===== *)
xHomeTrigY := HMI_xHomeY OR ((HMI_iHomeAxis = 1) AND HMI_xHomeExec);
xHomeTrigZ := HMI_xHomeZ OR ((HMI_iHomeAxis = 2) AND HMI_xHomeExec);
xHomeTrigR := HMI_xHomeR OR ((HMI_iHomeAxis = 3) AND HMI_xHomeExec);
xAnyHomeBusy := AxisCmd_xHomeY OR AxisCmd_xHomeZ OR AxisCmd_xHomeR;

IF AxisCmd_xStopAll OR NOT xSafe OR xFaultAggregate THEN
    AxisCmd_xHomeY := FALSE;
    AxisCmd_xHomeZ := FALSE;
    AxisCmd_xHomeR := FALSE;
ELSE
    IF AxisCmd_xHomeY AND AxisFb_xHomedY THEN AxisCmd_xHomeY := FALSE; END_IF;
    IF AxisCmd_xHomeZ AND AxisFb_xHomedZ THEN AxisCmd_xHomeZ := FALSE; END_IF;
    IF AxisCmd_xHomeR AND AxisFb_xHomedR THEN AxisCmd_xHomeR := FALSE; END_IF;
    IF (eOpMode = 0) AND NOT HMI_xStop THEN
        IF xHomeTrigY AND NOT xHomeTrigYPrev AND NOT xAnyHomeBusy THEN
            AxisCmd_xHomeY := TRUE;
        ELSIF xHomeTrigZ AND NOT xHomeTrigZPrev AND NOT xAnyHomeBusy THEN
            AxisCmd_xHomeZ := TRUE;
        ELSIF xHomeTrigR AND NOT xHomeTrigRPrev AND NOT xAnyHomeBusy AND xM5Ready THEN
            AxisCmd_xHomeR := TRUE;
        END_IF;
    END_IF;
END_IF;
xHomeTrigYPrev := xHomeTrigY;
xHomeTrigZPrev := xHomeTrigZ;
xHomeTrigRPrev := xHomeTrigR;

IF AxisCmd_xHomeY THEN xCmdJogYPos := FALSE; xCmdJogYNeg := FALSE; END_IF;
IF AxisCmd_xHomeZ THEN xCmdJogZPos := FALSE; xCmdJogZNeg := FALSE; xCmdForceFollow := FALSE; END_IF;
IF AxisCmd_xHomeR THEN xCmdJogRPos := FALSE; xCmdJogRNeg := FALSE; END_IF;

(* 本扫描只写一次 GVL，ETHERCAT 不会采到中途 FALSE *)
AxisCmd_xJogXPos := xCmdJogXPos; AxisCmd_xJogXNeg := xCmdJogXNeg;
AxisCmd_xSpinLeft := xCmdSpinL; AxisCmd_xSpinRight := xCmdSpinR;
AxisCmd_xJogYPos := xCmdJogYPos; AxisCmd_xJogYNeg := xCmdJogYNeg;
AxisCmd_xJogZPos := xCmdJogZPos; AxisCmd_xJogZNeg := xCmdJogZNeg;
AxisCmd_xJogRPos := xCmdJogRPos; AxisCmd_xJogRNeg := xCmdJogRNeg;
AxisCmd_xForceFollow := xCmdForceFollow;
AxisCmd_xMoveRelX := xCmdMoveRelX;
AxisCmd_xMoveRelY := xCmdMoveRelY;
AxisCmd_xMoveAbsY := xCmdMoveAbsY;
AxisCmd_xHoldR := xCmdHoldR;
(* 0.68 全轴直控：模式仲裁结果一次性写 AxisCmd_*，避免同扫描 TRUE->FALSE 空窗 *)
AxisCmd_xDirectVelY := xDirectVelY; AxisCmd_xDirectVelZ := xDirectVelZ; AxisCmd_xDirectVelR := xDirectVelR;
AxisCmd_xDirectAbsY := xDirectAbsY; AxisCmd_xDirectAbsZ := xDirectAbsZ; AxisCmd_xDirectAbsR := xDirectAbsR;
AxisCmd_xDirectRelY := xDirectRelY; AxisCmd_xDirectRelZ := xDirectRelZ; AxisCmd_xDirectRelR := xDirectRelR;
AxisCmd_rDirectVelY := rDirectVelYSel; AxisCmd_rDirectVelZ := rDirectVelZSel; AxisCmd_rDirectVelR := rDirectVelRSel;
AxisCmd_rDirectAbsY := rDirectPosYSel; AxisCmd_rDirectAbsZ := rDirectPosZSel; AxisCmd_rDirectAbsR := rDirectPosRSel;
AxisCmd_rDirectRelY := rDirectPosYSel; AxisCmd_rDirectRelZ := rDirectPosZSel; AxisCmd_rDirectRelR := rDirectPosRSel;

HMI_xHomedY := AxisFb_xHomedY;
HMI_xHomedZ := AxisFb_xHomedZ;
HMI_xHomedR := AxisFb_xHomedR;
HMI_xHomeBusyY := AxisCmd_xHomeY;
HMI_xHomeBusyZ := AxisCmd_xHomeZ;
HMI_xHomeBusyR := AxisCmd_xHomeR;

(* 使能就绪诊断 → 1007 *)
xReadyAll := AxisFb_xReadyM1 AND AxisFb_xReadyM2 AND AxisFb_xReadyY AND AxisFb_xReadyZ
    AND (NOT xM5Ready OR AxisFb_xReadyR);
tonReady(IN := AxisCmd_xPower AND NOT xReadyAll AND NOT xFaultAggregate, PT := T#2S);

(* 报警 *)
IF xEStopLatched OR NOT HMI_xEStop THEN
    iAlarmID := 1001;
ELSIF AxisFb_xFaultM1 OR AxisFb_xFaultM2 OR AxisFb_xFaultY OR AxisFb_xFaultZ
        OR (xM5Ready AND AxisFb_xFaultR) THEN
    iAlarmID := 1002;
ELSIF tonReady.Q THEN
    iAlarmID := 1007;
ELSIF NOT HMI_xForceSimEnable AND Force_xSlaveFail THEN
    iAlarmID := 1006;
ELSIF NOT HMI_xForceSimEnable AND Force_xTimeout THEN
    iAlarmID := 1005;
ELSE
    iAlarmID := 0;
END_IF;

(* 状态灯（只读派生，不互锁） *)
Dev_xError := xFaultAggregate;
Dev_xRun := xSafe AND NOT HMI_xStop AND NOT xFaultAggregate;
Dev_xStop := NOT Dev_xRun AND NOT Dev_xError;
HMI_xDevError := Dev_xError;
HMI_xDevRun := Dev_xRun;
HMI_xDevStop := Dev_xStop;
IF Dev_xError THEN HMI_eDevState := 2;
ELSIF Dev_xRun THEN HMI_eDevState := 1;
ELSE HMI_eDevState := 0; END_IF;

HMI_iAutoStepShow := iAutoStep;
HMI_xLampEStop := xEStopLatched OR NOT HMI_xEStop;
HMI_xLampEnableOk := Dev_xRun;
HMI_xLampFault := xFaultAggregate;
HMI_iAlarmShow := iAlarmID;

StopLamp := Dev_xStop;
StartLamp := Dev_xRun;
          
END_PROGRAM

PROGRAM PRG_Force485
  VAR
    iSlaveStep : INT;
    iSlaveTry : INT;
    tonSlave : TON;
    wSnap : WORD;
    wRawLast : WORD;
    xTarePrev : BOOL;
    xUntarePrev : BOOL;
    xUnitInit : BOOL;
    diRaw : DINT;
    rTmp : REAL;
    xTareReq : BOOL;
  END_VAR

            (*==============================================================================
 * PRG_Force485 — SM1001 使能 + 发读等回文（最多3次）+ 去皮/换算
 *
 * 流程（严格按需求）：
 *   1) 使能 Modbus 从站 SM1001
 *   2) 发送一次读（破坏 Force_wInRaw 快照，等组态 FC03 通道写回 = 有回文）
 *   3) 有回文 → Force_xCommOk，进入成功态，不再重试
 *   4) 无回文 → 关闭 SM1001，重新使能，再读
 *   5) 3 次均无回文 → Force_xSlaveFail / 报警 1006
 *
 * 组态：读通道 FC03 0x0000 → Force_wInRaw（循环或由 Force_xReadTrig 触发均可）
 *============================================================================*)

Force_xTareDone := FALSE;

IF NOT Force_xEnable THEN
	SM1001 := FALSE;
	Force_xReadTrig := FALSE;
	Force_xCommOk := FALSE;
	Force_xTimeout := FALSE;
	Force_xTareBusy := FALSE;
	Force_xSlaveFail := FALSE;
	Force_iState := 0;
	iSlaveStep := 0;
	iSlaveTry := 0;
	RETURN;
END_IF;

CASE iSlaveStep OF
	0: (* 准备：先关从站，再进入使能 *)
		IF iSlaveTry >= 3 THEN
			SM1001 := FALSE;
			Force_xReadTrig := FALSE;
			Force_xSlaveFail := TRUE;
			Force_xTimeout := TRUE;
			Force_xCommOk := FALSE;
			Force_iState := -2;
			iSlaveStep := 99;
		ELSE
			SM1001 := FALSE;
			Force_xReadTrig := FALSE;
			Force_xCommOk := FALSE;
			tonSlave(IN := FALSE);
			tonSlave(IN := TRUE, PT := T#200MS);
			Force_iState := 0;
			iSlaveStep := 1;
		END_IF;

	1: (* 关断保持 *)
		SM1001 := FALSE;
		Force_xReadTrig := FALSE;
		tonSlave();
		IF tonSlave.Q THEN
			tonSlave(IN := FALSE);
			iSlaveStep := 2;
		END_IF;

	2: (* ① 使能从站 *)
		SM1001 := TRUE;
		Force_xReadTrig := FALSE;
		iSlaveTry := iSlaveTry + 1;
		tonSlave(IN := FALSE);
		tonSlave(IN := TRUE, PT := T#100MS);
		Force_iState := 1;
		iSlaveStep := 3;

	3: (* 使能稳定后：② 发读命令（破坏快照 + 读触发） *)
		SM1001 := TRUE;
		tonSlave();
		IF tonSlave.Q THEN
			(* 破坏映射值：有回文时通道会写回真实寄存器 *)
			wSnap := Force_wInRaw XOR 16#FFFF;
			Force_wInRaw := wSnap;
			Force_xReadTrig := FALSE;
			tonSlave(IN := FALSE);
			tonSlave(IN := TRUE, PT := T#20MS);
			Force_iState := 2;
			iSlaveStep := 4;
		END_IF;

	4: (* 读触发上升沿 *)
		SM1001 := TRUE;
		tonSlave();
		IF tonSlave.Q THEN
			Force_xReadTrig := TRUE;
			tonSlave(IN := FALSE);
			tonSlave(IN := TRUE, PT := T#500MS);
			Force_iState := 3;
			iSlaveStep := 5;
		END_IF;

	5: (* ③ 等回文：Force_wInRaw 被总线写回且不等于破坏值 *)
		SM1001 := TRUE;
		Force_xReadTrig := TRUE;
		tonSlave();
		IF Force_wInRaw <> wSnap THEN
			(* 有回文 → 成功，不再尝试 *)
			Force_xReadTrig := FALSE;
			Force_xCommOk := TRUE;
			Force_xTimeout := FALSE;
			Force_xSlaveFail := FALSE;
			wRawLast := Force_wInRaw;
			Force_iState := 4;
			tonSlave(IN := FALSE);
			iSlaveStep := 10;
		ELSIF tonSlave.Q THEN
			(* 无回文 → 关从站，回到 0 重新使能 *)
			Force_xReadTrig := FALSE;
			SM1001 := FALSE;
			Force_xCommOk := FALSE;
			Force_iState := 5;
			tonSlave(IN := FALSE);
			iSlaveStep := 0;
		END_IF;

	10: (* 成功：保持使能，不再重试使能 *)
		SM1001 := TRUE;
		Force_xReadTrig := FALSE;
		Force_xCommOk := TRUE;
		Force_xTimeout := FALSE;
		IF Force_wInRaw <> wRawLast THEN
			wRawLast := Force_wInRaw;
		END_IF;

	99: (* 3 次失败；复位清 Force_xSlaveFail 后从 0 重来 *)
		SM1001 := FALSE;
		Force_xReadTrig := FALSE;
		IF Force_xSlaveFail THEN
			Force_xTimeout := TRUE;
			Force_xCommOk := FALSE;
		ELSE
			iSlaveTry := 0;
			Force_xTimeout := FALSE;
			iSlaveStep := 0;
		END_IF;
END_CASE;

(* ----- 原始值换算（成功后持续；探测中也换算便于监视） ----- *)
diRaw := DWORD_TO_DINT(WORD_TO_DWORD(Force_wInRaw));
IF diRaw > 32767 THEN
	diRaw := diRaw - 65536;
END_IF;
Force_iRaw := DINT_TO_INT(diRaw);
IF Force_rScale < 1.0E-12 THEN
	rTmp := INT_TO_REAL(Force_iRaw);
ELSE
	rTmp := INT_TO_REAL(Force_iRaw) * Force_rScale;
END_IF;
IF NOT HMI_xForceSimEnable AND iSlaveStep = 10 THEN
	rForceAct := rTmp;
END_IF;

IF NOT xUnitInit AND iSlaveStep = 10 THEN
	Force_wOutUnit := 5;
	xUnitInit := TRUE;
END_IF;

xTareReq := FALSE;
IF iSlaveStep = 10 THEN
	IF ((HMI_xForceTare OR Tcp_xForceTare OR Logic_xForceTare) AND NOT xTarePrev) THEN
		Force_wOutTare := 1;
		xTareReq := TRUE;
		Force_xTareDone := TRUE;
	END_IF;
	xTarePrev := HMI_xForceTare OR Tcp_xForceTare OR Logic_xForceTare;
	IF Tcp_xForceTare THEN
		Tcp_xForceTare := FALSE;
	END_IF;
	IF Logic_xForceTare THEN
		Logic_xForceTare := FALSE;
	END_IF;

	IF ((HMI_xForceUntare OR Tcp_xForceUntare) AND NOT xUntarePrev) THEN
		Force_wOutTare := 2;
		xTareReq := TRUE;
		Force_xTareDone := TRUE;
	END_IF;
	xUntarePrev := HMI_xForceUntare OR Tcp_xForceUntare;
	IF Tcp_xForceUntare THEN
		Tcp_xForceUntare := FALSE;
	END_IF;
END_IF;

Force_xTareBusy := xTareReq;

          
END_PROGRAM

FUNCTION_BLOCK FB_Servo
  VAR_INPUT
    xEnable : BOOL;  (* 驱动器使能（来自 AxisCmd_xPower） *)
    xStop : BOOL;  (* 停止运动（保持使能） *)
    xResetFault : BOOL;  (* 故障复位（上升沿） *)
    xHome : BOOL;  (* 回零（电平，完成/撤销后由上层清） *)
    xMoveAbs : BOOL;  (* 绝对定位（电平保持至完成） *)
    rTargetPos : REAL;  (* 绝对目标位置 *)
    xMoveRel : BOOL;  (* 相对定位（电平保持至完成） *)
    rDist : REAL;  (* 相对距离（可正可负） *)
    xUseVelCmd : BOOL;  (* 速度指令模式（力跟随/X双驱） *)
    rVelCmd : REAL;  (* 速度给定（可正可负；|v|<1e-6 视为撤销） *)
    xJogPos : BOOL;  (* 点动+（电平，MC_Jog） *)
    xJogNeg : BOOL;  (* 点动-（电平，MC_Jog） *)
    rJogVel : REAL;  (* 点动速度（正值） *)
    rVel : REAL;  (* 定位速度（正值） *)
    rAcc : REAL;  (* 加速度 *)
    rDec : REAL;  (* 减速度 *)
    xLimEn : BOOL;  (* 硬限位使能（X=FALSE，Y/Z/R=TRUE） *)
    rLimPos : REAL;  (* 正方向硬限位（可手动改） *)
    rLimNeg : REAL;  (* 负方向硬限位（可手动改） *)
  END_VAR
  VAR_OUTPUT
    xPowered : BOOL;  (* 驱动器已上电 := fbPower.Status *)
    xReady : BOOL;  (* 就绪 := 上电且无故障 *)
    xMoving : BOOL;  (* 运动中（含回零） *)
    xStandstill : BOOL;  (* 静止 *)
    xHomed : BOOL;  (* 回零完成（置零后保持） *)
    xFault : BOOL;  (* 故障 := MC_ReadStatus.ErrorStop *)
    xMoveRelDone : BOOL;  (* 相对定位完成 *)
    xMoveAbsDone : BOOL;  (* 绝对定位完成 *)
    rActPos : LREAL;  (* 实际位置 *)
    rVelAct : REAL;  (* 实际速度；g 线 0.68 直控/回读专用 *)
    xVelReq : BOOL;  (* 诊断：仲裁后速度请求已成立 *)
    xVelBusy : BOOL;  (* 诊断：MC_MoveVelocity.Busy *)
    xVelInVel : BOOL;  (* 诊断：MC_MoveVelocity.InVelocity *)
    xErrPower : BOOL;  (* 诊断：MC_Power.Error（驱动未就绪/通讯异常） *)
    xErrVel : BOOL;  (* 诊断：MC_MoveVelocity.Error（参数/平台拒绝） *)
    xErrJog : BOOL;  (* 诊断：MC_Jog.Error *)
    xErrHalt : BOOL;  (* 诊断：MC_Halt.Error *)
    xErrHome : BOOL;  (* 诊断：MC_Home.Error *)
    xErrAbs : BOOL;  (* 诊断：MC_MoveAbsolute.Error *)
    xErrRel : BOOL;  (* 诊断：MC_MoveRelative.Error *)
  END_VAR
  VAR
    fbPower : MC_Power;
    fbHalt : MC_Halt;
    fbHome : MC_Home;
    fbReset : MC_Reset;
    fbReadStatus : MC_ReadStatus;
    fbReadPos : MC_ReadActualPosition;
    fbSetPos : MC_SetPosition;
    fbMoveRel : MC_MoveRelative;
    fbMoveAbs : MC_MoveAbsolute;
    fbMoveVel : MC_MoveVelocity;
    fbJog : MC_Jog;
    eDir : MC_DIRECTION;
    xReqStop : BOOL;
    xReqHome : BOOL;
    xReqAbs : BOOL;
    xReqRel : BOOL;
    xReqVel : BOOL;
    xReqJogPos : BOOL;
    xReqJogNeg : BOOL;
    xReqAny : BOOL;
    xReqHomePrev : BOOL;
    xSetZeroTrig : BOOL;
    xVelRunPrev : BOOL;
    xDirFlip : BOOL;
    xNeedStop : BOOL;
    xHaltPrev : BOOL;
    xResetPrev : BOOL;
    xBlockPos : BOOL;
    xBlockNeg : BOOL;
    rAbsTarget : REAL;
    rRelDist : REAL;
    rVelInPrev : REAL;
  END_VAR
  VAR_IN_OUT
    Axis : AXIS_REF_SM3;
  END_VAR

            (* =============================================================================
   FB_Servo — 单轴原子封装（SM3_Basic）。仅在 PRG_Axis_Control 任务内实例化。

   仲裁优先级：停止/故障 > 回零 > 绝对定位 > 相对定位 > 速度指令 > 点动。
   - 手动点动走 MC_Jog（松开即减速停）；速度指令走 MC_MoveVelocity
   - 运动切换靠 PLCopen 中止机制（新命令 FB 上升沿自动 abort 旧运动）
   - 全部运动请求撤销（松手/速度归零/停止/急停/撞限位）→ MC_Halt 减速停车
   - 硬限位：xLimEn=TRUE 时，所有模式都限制在 [rLimNeg, rLimPos] 内：
     点动/速度 越限方向被禁止；定位目标被夹紧；X 轴传 xLimEn:=FALSE
   ========================================================================== *)

(* 1. 状态与位置 *)
fbReadStatus(Axis := Axis, Enable := TRUE);
fbReadPos(Axis := Axis, Enable := TRUE);
rActPos := fbReadPos.Position;
rVelAct := LREAL_TO_REAL(Axis.fActVelocity);
xStandstill := fbReadStatus.StandStill;
xFault := fbReadStatus.ErrorStop;
xMoving := fbReadStatus.DiscreteMotion OR fbReadStatus.ContinuousMotion OR fbReadStatus.Homing;

(* 2. 故障复位（上升沿） *)
fbReset(Axis := Axis, Execute := xResetFault AND NOT xResetPrev);
xResetPrev := xResetFault;

(* 3. 驱动器使能（xStop 不掉使能） *)
fbPower(Axis := Axis, Enable := TRUE,
        bRegulatorOn := xEnable AND NOT xFault,
        bDriveStart := xEnable AND NOT xFault);
xPowered := fbPower.Status;
xReady := xPowered AND NOT xFault;

(* 4. 硬限位：越限方向禁止；定位目标夹紧（已越限时仍允许向回运动） *)
xBlockPos := xLimEn AND (rActPos >= rLimPos);
xBlockNeg := xLimEn AND (rActPos <= rLimNeg);
rAbsTarget := rTargetPos;
rRelDist := rDist;
IF xLimEn THEN
    rAbsTarget := LIMIT(rLimNeg, rTargetPos, rLimPos);
    rRelDist := LIMIT(rLimNeg, rActPos + rDist, rLimPos) - rActPos;
END_IF;

(* 5. 命令仲裁：停止/故障 > 回零 > 绝对 > 相对 > 速度 > 点动 *)
xReqStop := xStop OR NOT xEnable OR xFault;
xReqHome := xHome AND NOT xReqStop;
xReqAbs := xMoveAbs AND xPowered AND NOT xReqStop AND NOT xReqHome;
xReqRel := xMoveRel AND (ABS(rRelDist) > 1.0E-9) AND xPowered
           AND NOT xReqStop AND NOT xReqHome AND NOT xReqAbs;
xReqVel := xUseVelCmd AND (ABS(rVelCmd) > 1.0E-6) AND xPowered
           AND NOT ((rVelCmd > 0.0) AND xBlockPos) AND NOT ((rVelCmd < 0.0) AND xBlockNeg)
           AND NOT xReqStop AND NOT xReqHome AND NOT xReqAbs AND NOT xReqRel;
xReqJogPos := xJogPos AND NOT xJogNeg AND NOT xBlockPos AND xPowered
              AND NOT xReqStop AND NOT xReqHome AND NOT xReqAbs AND NOT xReqRel AND NOT xReqVel;
xReqJogNeg := xJogNeg AND NOT xJogPos AND NOT xBlockNeg AND xPowered
              AND NOT xReqStop AND NOT xReqHome AND NOT xReqAbs AND NOT xReqRel AND NOT xReqVel;
xReqAny := xReqHome OR xReqAbs OR xReqRel OR xReqVel OR xReqJogPos OR xReqJogNeg;

(* 6. 回零：MC_Home(0) → MC_SetPosition(0) → xHomed *)
IF xReqHome AND NOT xReqHomePrev THEN
    xHomed := FALSE;
END_IF;
xReqHomePrev := xReqHome;
fbHome(Axis := Axis, Execute := xReqHome, Position := 0.0);
IF fbHome.Done THEN
    xSetZeroTrig := TRUE;
END_IF;
fbSetPos(Axis := Axis, Execute := xSetZeroTrig, Position := 0.0);
IF fbSetPos.Done THEN
    xHomed := TRUE;
    xSetZeroTrig := FALSE;
END_IF;

(* 7. 绝对 / 相对定位（目标已夹紧；电平保持 Execute，Done 上报） *)
fbMoveAbs(Axis := Axis, Execute := xReqAbs, Position := rAbsTarget,
          Velocity := ABS(rVel), Acceleration := rAcc, Deceleration := rDec);
fbMoveRel(Axis := Axis, Execute := xReqRel, Distance := rRelDist,
          Velocity := ABS(rVel), Acceleration := rAcc, Deceleration := rDec);
xMoveAbsDone := fbMoveAbs.Done;
xMoveRelDone := fbMoveRel.Done;

(* 8. 速度指令：MC_MoveVelocity；Velocity 取绝对值，方向走 Direction *)
(* 注意：本机 SM3 库的方向字面值是 positive/negative（非 CoDeSys 的 mcPositiveDirection） *)
IF rVelCmd >= 0.0 THEN
    eDir := positive;
ELSE
    eDir := negative;
END_IF;
(* 运行中换向：先撤 Execute 一拍，下一拍带新方向重新触发 *)
xDirFlip := xReqVel AND xVelRunPrev AND ((rVelCmd >= 0.0) <> (rVelInPrev >= 0.0));
fbMoveVel(Axis := Axis, Execute := xReqVel AND NOT xDirFlip,
          Velocity := ABS(rVelCmd), Direction := eDir,
          Acceleration := rAcc, Deceleration := rDec);
xVelRunPrev := xReqVel;
rVelInPrev := rVelCmd;

(* 9. 手动点动：MC_Jog（按住动、松开减速停；越限方向已在仲裁禁止） *)
fbJog(Axis := Axis,
      JogForward := xReqJogPos,
      JogBackward := xReqJogNeg,
      Velocity := ABS(rJogVel),
      Acceleration := rAcc,
      Deceleration := rDec);

(* 10. 停车：有使能但无任何运动请求（松手/速度归零/停止/急停/撞限位）→ MC_Halt *)
xNeedStop := xPowered AND NOT xReqAny;
fbHalt(Axis := Axis, Execute := xNeedStop AND xMoving AND NOT xHaltPrev,
       Deceleration := rDec);
xHaltPrev := xNeedStop AND xMoving;

(* 11. 诊断输出（g 线 0.5） *)
xVelReq := xReqVel;
xVelBusy := fbMoveVel.Busy;
xVelInVel := fbMoveVel.InVelocity;
xErrPower := fbPower.Error;
xErrVel := fbMoveVel.Error;
xErrJog := fbJog.Error;
xErrHalt := fbHalt.Error;
xErrHome := fbHome.Error;
xErrAbs := fbMoveAbs.Error;
xErrRel := fbMoveRel.Error;
          
END_FUNCTION_BLOCK

FUNCTION_BLOCK FB_Force
  VAR_INPUT
    wRaw : WORD;  (* 组态映射原始力 %IW102 *)
    rScale : REAL;  (* 倍率，默认 0.01 *)
    xEnable : BOOL;  (* 通讯总使能 *)
    xTare : BOOL;  (* 去皮（上升沿记偏移） *)
    xUntare : BOOL;  (* 取消去皮（上升沿清偏移） *)
  END_VAR
  VAR_OUTPUT
    rForceN : REAL;  (* 实际力 N *)
    iRaw : INT;  (* 有符号原始计数 *)
    xCommOk : BOOL;  (* 通讯正常 *)
    xTimeout : BOOL;  (* 2s 原始值不变 → 超时（报警 1005） *)
  END_VAR
  VAR
    rTare : REAL;
    xTarePrev : BOOL;
    xUntarePrev : BOOL;
    wPrev : WORD;
    tonStale : TON;
    rRawScaled : REAL;
  END_VAR

            (* FB_Force — Modbus 原始力换算 + 软件去皮 + 通讯看门狗（仅提示，不进故障） *)

iRaw := WORD_TO_INT(wRaw);
rRawScaled := INT_TO_REAL(iRaw) * rScale;

IF xTare AND NOT xTarePrev THEN
    rTare := rRawScaled;
END_IF;
xTarePrev := xTare;
IF xUntare AND NOT xUntarePrev THEN
    rTare := 0.0;
END_IF;
xUntarePrev := xUntare;

rForceN := rRawScaled - rTare;

tonStale(IN := xEnable AND (wRaw = wPrev), PT := T#2S);
wPrev := wRaw;
xTimeout := xEnable AND tonStale.Q;
xCommOk := xEnable AND NOT xTimeout;
          
END_FUNCTION_BLOCK

FUNCTION_BLOCK FB_ForceFollow
  VAR_INPUT
    rForceSet : REAL;  (* 目标力 N *)
    rForceAct : REAL;  (* 实际力 N *)
    rKp : REAL;  (* 比例增益，越大响应越快，过大易抖 *)
    rVelMax : REAL;  (* 速度限幅（正值） *)
    rDeadband : REAL;  (* 死区 N，区内输出 0 *)
    rPosZ : LREAL;  (* Z 实际位置 *)
    rLimPos : REAL;  (* Z 正限位（同 Cfg_rLimZPos） *)
    rLimNeg : REAL;  (* Z 负限位（同 Cfg_rLimZNeg） *)
    xEnable : BOOL;  (* 力跟随使能（电平） *)
    xInvert : BOOL;  (* 现场方向翻转 *)
  END_VAR
  VAR_OUTPUT
    rZVelCmd : REAL;  (* Z 速度指令输出 *)
    xInBand : BOOL;  (* 力在死区内 *)
  END_VAR
  VAR
    rErr : REAL;
    rV : REAL;
  END_VAR

            (* FB_ForceFollow — Z 恒力 P 控制律；向下=负增压；硬限位 [rLimNeg, rLimPos] 内跟随 *)

IF NOT xEnable THEN
    rZVelCmd := 0.0;
    xInBand := FALSE;
    RETURN;
END_IF;

rErr := rForceSet - rForceAct;
rV := -rKp * rErr;
IF xInvert THEN
    rV := -rV;
END_IF;
rV := LIMIT(-ABS(rVelMax), rV, ABS(rVelMax));

xInBand := ABS(rErr) < rDeadband;
IF xInBand THEN
    rV := 0.0;
END_IF;

(* 硬限位：越限方向输出 0（FB_Servo 另有最终闸门） *)
IF (rPosZ >= rLimPos) AND (rV > 0.0) THEN
    rV := 0.0;
END_IF;
IF (rPosZ <= rLimNeg) AND (rV < 0.0) THEN
    rV := 0.0;
END_IF;

rZVelCmd := rV;
          
END_FUNCTION_BLOCK

PROGRAM PRG_Axis_Control
  VAR
    fbX : FB_XDual;
    fbY : FB_Servo;
    fbZ : FB_Servo;
    fbR : FB_Servo;
    fbForce : FB_Force;
    fbFF : FB_ForceFollow;
  END_VAR

            (* PRG_Axis_Control — 运动独立任务(ETHERCAT 4ms)。只读 AxisCmd_*，写 AxisFb_*/rForceAct。
   禁止被其它 POU CALL；禁止写 HMI_*/报警。
   X：FB_XDual（LineTrack + 双 FB_Servo，无 Virtual/Gear）；Y/Z/R 仍 FB_Servo。 *)

(* ===== 力传感转换（本 POU 拥有 rForceAct） ===== *)
fbForce(wRaw := Force_wInRaw, rScale := Force_rScale, xEnable := Force_xEnable,
    xTare := HMI_xForceTare OR Logic_xForceTare, xUntare := HMI_xForceUntare);
Force_iRaw := fbForce.iRaw;
(* 力通讯状态由 PRG_Force485 的收发回文状态机唯一判定；
   不再用 FB_Force 的“原始值 2s 不变”看门狗覆盖，避免力稳定时误报 1005。 *)
IF NOT HMI_xForceSimEnable THEN
    rForceAct := fbForce.rForceN;
END_IF;

(* ===== X：FB_XDual（LineTrack + 双 Servo；无 Virtual/Gear） ===== *)
fbX(
    AxisM1 := Axis, AxisM2 := Axis_1,
    xEnable := AxisCmd_xPower, xStop := AxisCmd_xStopAll, xResetFault := AxisCmd_xResetFault,
    xJogPos := AxisCmd_xJogXPos, xJogNeg := AxisCmd_xJogXNeg,
    xSpinLeft := AxisCmd_xSpinLeft, xSpinRight := AxisCmd_xSpinRight,
    xMoveRel := AxisCmd_xMoveRelX, rMoveDist := AxisCmd_rMoveDistX, rMoveVel := AxisCmd_rMoveVelX,
    rJogVel := AxisCmd_rJogVelX, rSpinVel := AxisCmd_rSpinVel,
    rHeadingErr := AxisCmd_rHeadingErr, rKpTrack := AxisCmd_rTrackKp,
    rAcc := AxisCmd_rAccX, rDec := AxisCmd_rDecX,
    rTrimMax := Cfg_rPhaseMax,
    (* 0.60 视觉直控：绕过内部差速，直接给 M1/M2 速度 *)
    xDirectMode := AxisCmd_xDirectVel,
    rVelM1Direct := AxisCmd_rVelM1Set, rVelM2Direct := AxisCmd_rVelM2Set,
    wSdoDevM1 := Cfg_wSdoDevM1, wSdoDevM2 := Cfg_wSdoDevM2,
    xForceCsv := Cfg_xForceCsvX);
AxisFb_xMoveDoneX := fbX.xMoveDone;
AxisFb_rPosX := fbX.rPosV;
AxisFb_rSyncErr := fbX.rSyncErr;
AxisFb_rVelFactorX := fbX.rVelFactor;
AxisFb_xGantryCoupled := fbX.xCoupled;
AxisFb_xInGearM1 := fbX.xInGearM1;
AxisFb_xInGearM2 := fbX.xInGearM2;
AxisFb_xPoweredV := fbX.xPoweredV;
AxisFb_xSyncWarn := fbX.xSyncWarn;
AxisFb_xSyncFault := fbX.xSyncFault;
AxisFb_iGantryState := fbX.iState;
AxisFb_rVelCmdM1 := fbX.rVelCmdM1;
AxisFb_rVelCmdM2 := fbX.rVelCmdM2;
(* 0.71 M1/M2 转矩/电流（CoE 0x6077/0x6078 慢速读取，‰额定） *)
AxisFb_rTorqueM1 := fbX.rTorqueActM1;
AxisFb_rTorqueM2 := fbX.rTorqueActM2;
AxisFb_rCurrentM1 := fbX.rCurrentActM1;
AxisFb_rCurrentM2 := fbX.rCurrentActM2;
AxisFb_xParamErr := fbX.xParamErr;
(* 0.72 驱动诊断（原始 16 位） *)
AxisFb_wSwM1 := fbX.wSwM1;
AxisFb_wErrM1 := fbX.wErrM1;
AxisFb_wTqMaxM1 := fbX.wTqMaxM1;
AxisFb_wLimPM1 := fbX.wLimPM1;
AxisFb_wLimNM1 := fbX.wLimNM1;
AxisFb_wSwM2 := fbX.wSwM2;
AxisFb_wErrM2 := fbX.wErrM2;
AxisFb_wTqMaxM2 := fbX.wTqMaxM2;
AxisFb_wLimPM2 := fbX.wLimPM2;
AxisFb_wLimNM2 := fbX.wLimNM2;
(* 0.73 MDX：模式(0x6060) + 转矩限值(0x2403~0x2406) *)
AxisFb_wModeM1 := fbX.wModeM1;
AxisFb_wTq03M1 := fbX.wTq03M1;
AxisFb_wTq04M1 := fbX.wTq04M1;
AxisFb_wTq05M1 := fbX.wTq05M1;
AxisFb_wTq06M1 := fbX.wTq06M1;
AxisFb_wModeM2 := fbX.wModeM2;
AxisFb_wTq03M2 := fbX.wTq03M2;
AxisFb_wTq04M2 := fbX.wTq04M2;
AxisFb_wTq05M2 := fbX.wTq05M2;
AxisFb_wTq06M2 := fbX.wTq06M2;
(* 0.74 CSV 模式切换状态 *)
AxisFb_xModeCsvM1 := fbX.xModeCsvM1;
AxisFb_xModeCsvErrM1 := fbX.xModeCsvErrM1;
AxisFb_xModeCsvM2 := fbX.xModeCsvM2;
AxisFb_xModeCsvErrM2 := fbX.xModeCsvErrM2;
AxisFb_rPosM1 := fbX.rPosM1;
AxisFb_rPosM2 := fbX.rPosM2;
AxisFb_xMovingM1 := fbX.xMovingM1;
AxisFb_xMovingM2 := fbX.xMovingM2;
AxisFb_xStandstill1 := fbX.xStandstillM1;
AxisFb_xStandstill2 := fbX.xStandstillM2;
AxisFb_xPoweredM1 := fbX.xPoweredM1;
AxisFb_xPoweredM2 := fbX.xPoweredM2;
AxisFb_xReadyM1 := fbX.xReadyM1;
AxisFb_xReadyM2 := fbX.xReadyM2;
AxisFb_xFaultM1 := fbX.xFaultM1;
AxisFb_xFaultM2 := fbX.xFaultM2;

(* 0.60 视觉直控反馈（回给 PRG_TcpHmi 编码到状态镜像 + 视觉侧回读） *)
Direct_xActive := fbX.xDirectActive;
Direct_rVelM1Act := fbX.rVelActM1Out;
Direct_rVelM2Act := fbX.rVelActM2Out;

(* 0.63 通用双电机实际速度透传（供 PRG_TcpHmi 编码到状态 word32..38） *)
AxisFb_rVelActM1 := fbX.rVelActM1Out;
AxisFb_rVelActM2 := fbX.rVelActM2Out;

(* ===== Y：回零 > 绝对(归位) > 相对(横移) > 点动；硬限位 [Cfg_rLimYNeg, Cfg_rLimYPos] ===== *)
fbY(Axis := Axis_2, xEnable := AxisCmd_xPower, xStop := AxisCmd_xStopAll, xResetFault := AxisCmd_xResetFault,
    xHome := AxisCmd_xHomeY,
    xMoveAbs := AxisCmd_xMoveAbsY OR AxisCmd_xDirectAbsY,
    rTargetPos := SEL(AxisCmd_xMoveAbsY, AxisCmd_rDirectAbsY, AxisCmd_rMoveAbsPosY),
    xMoveRel := AxisCmd_xMoveRelY OR AxisCmd_xDirectRelY,
    rDist := SEL(AxisCmd_xMoveRelY, AxisCmd_rDirectRelY, AxisCmd_rMoveDistY),
    xUseVelCmd := AxisCmd_xDirectVelY, rVelCmd := AxisCmd_rDirectVelY,
    xJogPos := AxisCmd_xJogYPos, xJogNeg := AxisCmd_xJogYNeg, rJogVel := AxisCmd_rJogVelY,
    rVel := SEL(AxisCmd_xDirectAbsY OR AxisCmd_xDirectRelY, AxisCmd_rMoveVelY, AxisCmd_rDirectVelY),
    rAcc := AxisCmd_rAccY, rDec := AxisCmd_rDecY,
    xLimEn := TRUE, rLimPos := Cfg_rLimYPos, rLimNeg := Cfg_rLimYNeg);
AxisFb_xMoveDoneY := fbY.xMoveRelDone;

(* ===== Z：力跟随速度 > 回零 > 点动；硬限位 [Cfg_rLimZNeg, Cfg_rLimZPos] ===== *)
fbFF(rForceSet := AxisCmd_rForceSet, rForceAct := rForceAct, rKp := AxisCmd_rForceKp,
    rVelMax := AxisCmd_rForceVelMax, rDeadband := 0.5, rPosZ := fbZ.rActPos,
    rLimPos := Cfg_rLimZPos, rLimNeg := Cfg_rLimZNeg,
    xEnable := AxisCmd_xForceFollow, xInvert := FALSE);
fbZ(Axis := Axis_3, xEnable := AxisCmd_xPower, xStop := AxisCmd_xStopAll, xResetFault := AxisCmd_xResetFault,
    xHome := AxisCmd_xHomeZ,
    xMoveAbs := AxisCmd_xDirectAbsZ, rTargetPos := AxisCmd_rDirectAbsZ,
    xMoveRel := AxisCmd_xDirectRelZ, rDist := AxisCmd_rDirectRelZ,
    xUseVelCmd := AxisCmd_xForceFollow OR AxisCmd_xDirectVelZ,
    rVelCmd := SEL(AxisCmd_xForceFollow, AxisCmd_rDirectVelZ, fbFF.rZVelCmd),
    xJogPos := AxisCmd_xJogZPos, xJogNeg := AxisCmd_xJogZNeg, rJogVel := AxisCmd_rJogVelZ,
    rVel := AxisCmd_rDirectVelZ,
    rAcc := AxisCmd_rAccZ, rDec := AxisCmd_rDecZ,
    xLimEn := TRUE, rLimPos := Cfg_rLimZPos, rLimNeg := Cfg_rLimZNeg);

(* ===== R：回零 > 保持角(绝对) > 点动；M5 门控；硬限位 [Cfg_rLimRNeg, Cfg_rLimRPos] ===== *)
fbR(Axis := Axis_4, xEnable := AxisCmd_xPower AND xM5Ready, xStop := AxisCmd_xStopAll, xResetFault := AxisCmd_xResetFault,
    xHome := AxisCmd_xHomeR,
    xMoveAbs := AxisCmd_xHoldR OR AxisCmd_xDirectAbsR,
    rTargetPos := SEL(AxisCmd_xHoldR, AxisCmd_rDirectAbsR, AxisCmd_rRHoldPos),
    xMoveRel := AxisCmd_xDirectRelR, rDist := AxisCmd_rDirectRelR,
    xUseVelCmd := AxisCmd_xDirectVelR, rVelCmd := AxisCmd_rDirectVelR,
    xJogPos := AxisCmd_xJogRPos, xJogNeg := AxisCmd_xJogRNeg, rJogVel := AxisCmd_rJogVelR,
    rVel := SEL(AxisCmd_xDirectAbsR OR AxisCmd_xDirectRelR, AxisCmd_rJogVelR, AxisCmd_rDirectVelR),
    rAcc := AxisCmd_rAccR, rDec := AxisCmd_rDecR,
    xLimEn := TRUE, rLimPos := Cfg_rLimRPos, rLimNeg := Cfg_rLimRNeg);

(* ===== Y/Z/R 反馈回写 ===== *)
AxisFb_rPosY := fbY.rActPos; AxisFb_rPosZ := fbZ.rActPos; AxisFb_rPosR := fbR.rActPos;
AxisFb_xMovingY := fbY.xMoving; AxisFb_xMovingZ := fbZ.xMoving; AxisFb_xMovingR := fbR.xMoving;
AxisFb_xStandstillY := fbY.xStandstill; AxisFb_xStandstillZ := fbZ.xStandstill; AxisFb_xStandstillR := fbR.xStandstill;
AxisFb_xPoweredY := fbY.xPowered; AxisFb_xPoweredZ := fbZ.xPowered; AxisFb_xPoweredR := fbR.xPowered;
AxisFb_xReadyY := fbY.xReady; AxisFb_xReadyZ := fbZ.xReady; AxisFb_xReadyR := fbR.xReady;
AxisFb_xHomedY := fbY.xHomed; AxisFb_xHomedZ := fbZ.xHomed; AxisFb_xHomedR := fbR.xHomed;
AxisFb_xFaultY := fbY.xFault; AxisFb_xFaultZ := fbZ.xFault; AxisFb_xFaultR := fbR.xFault;
(* 0.68 全轴直控：Y/Z/R 实际速度回读（状态镜像 word39..41） *)
AxisFb_rVelActY := fbY.rVelAct;
AxisFb_rVelActZ := fbZ.rVelAct;
AxisFb_rVelActR := fbR.rVelAct;
AxisFb_xReady := AxisFb_xReadyM1 AND AxisFb_xReadyM2 AND fbY.xReady AND fbZ.xReady
    AND (NOT xM5Ready OR fbR.xReady);
          
END_PROGRAM

